   AxisStore[5].Axis[1..15].Pos26.Reached := FALSE;
   AxisStore[6].Axis[1..15].Pos26.Reached := FALSE;
   AxisStore[7].Axis[1..15].Pos26.Reached := FALSE;
   AxisStore[8].Axis[1..15].Pos26.Reached := FALSE;
   AxisStore[9].Axis[1..15].Pos26.Reached := FALSE;
   AxisStore[10].Axis[1..15].Pos26.Reached := FALSE;
   AxisStore[11].Axis[1..15].Pos26.Reached := FALSE;
   AxisStore[12].Axis[1..15].Pos26.Reached := FALSE;
   AxisStore[13].Axis[1..15].Pos26.Reached := FALSE;
   AxisStore[14].Axis[1..15].Pos26.Reached := FALSE;
   AxisStore[15].Axis[1..15].Pos26.Reached := FALSE;
   AxisStore[1].Axis[1..15].Pos27.Position := 0.0;
   AxisStore[2].Axis[1..15].Pos27.Position := 0.0;
   AxisStore[3].Axis[1..15].Pos27.Position := 0.0;
   AxisStore[4].Axis[1..15].Pos27.Position := 0.0;
   AxisStore[5].Axis[1..15].Pos27.Position := 0.0;
   AxisStore[6].Axis[1..15].Pos27.Position := 0.0;
   AxisStore[7].Axis[1..15].Pos27.Position := 0.0;
   AxisStore[8].Axis[1..15].Pos27.Position := 0.0;
   AxisStore[9].Axis[1..15].Pos27.Position := 0.0;
   AxisStore[10].Axis[1..15].Pos27.Position := 0.0;
   AxisStore[11].Axis[1..15].Pos27.Position := 0.0;
   AxisStore[12].Axis[1..15].Pos27.Position := 0.0;
   AxisStore[13].Axis[1..15].Pos27.Position := 0.0;
   AxisStore[14].Axis[1..15].Pos27.Position := 0.0;
   AxisStore[15].Axis[1..15].Pos27.Position := 0.0;
   AxisStore[1].Axis[1..15].Pos27.Speed := 0;
   AxisStore[2].Axis[1..15].Pos27.Speed := 0;
   AxisStore[3].Axis[1..15].Pos27.Speed := 0;
   AxisStore[4].Axis[1..15].Pos27.Speed := 0;
   AxisStore[5].Axis[1..15].Pos27.Speed := 0;
   AxisStore[6].Axis[1..15].Pos27.Speed := 0;
   AxisStore[7].Axis[1..15].Pos27.Speed := 0;
   AxisStore[8].Axis[1..15].Pos27.Speed := 0;
   AxisStore[9].Axis[1..15].Pos27.Speed := 0;
   AxisStore[10].Axis[1..15].Pos27.Speed := 0;
   AxisStore[11].Axis[1..15].Pos27.Speed := 0;
   AxisStore[12].Axis[1..15].Pos27.Speed := 0;
   AxisStore[13].Axis[1..15].Pos27.Speed := 0;
   AxisStore[14].Axis[1..15].Pos27.Speed := 0;
   AxisStore[15].Axis[1..15].Pos27.Speed := 0;
   AxisStore[1].Axis[1..15].Pos27.Reached := FALSE;
   AxisStore[2].Axis[1..15].Pos27.Reached := FALSE;
   AxisStore[3].Axis[1..15].Pos27.Reached := FALSE;
   AxisStore[4].Axis[1..15].Pos27.Reached := FALSE;
   AxisStore[5].Axis[1..15].Pos27.Reached := FALSE;
   AxisStore[6].Axis[1..15].Pos27.Reached := FALSE;
   AxisStore[7].Axis[1..15].Pos27.Reached := FALSE;
   AxisStore[8].Axis[1..15].Pos27.Reached := FALSE;
   AxisStore[9].Axis[1..15].Pos27.Reached := FALSE;
   AxisStore[10].Axis[1..15].Pos27.Reached := FALSE;
   AxisStore[11].Axis[1..15].Pos27.Reached := FALSE;
   AxisStore[12].Axis[1..15].Pos27.Reached := FALSE;
   AxisStore[13].Axis[1..15].Pos27.Reached := FALSE;
   AxisStore[14].Axis[1..15].Pos27.Reached := FALSE;
   AxisStore[15].Axis[1..15].Pos27.Reached := FALSE;
   AxisStore[1].Axis[1..15].Pos28.Position := 0.0;
   AxisStore[2].Axis[1..15].Pos28.Position := 0.0;
   AxisStore[3].Axis[1..15].Pos28.Position := 0.0;
   AxisStore[4].Axis[1..15].Pos28.Position := 0.0;
   AxisStore[5].Axis[1..15].Pos28.Position := 0.0;
   AxisStore[6].Axis[1..15].Pos28.Position := 0.0;
   AxisStore[7].Axis[1..15].Pos28.Position := 0.0;
   AxisStore[8].Axis[1..15].Pos28.Position := 0.0;
   AxisStore[9].Axis[1..15].Pos28.Position := 0.0;
   AxisStore[10].Axis[1..15].Pos28.Position := 0.0;
   AxisStore[11].Axis[1..15].Pos28.Position := 0.0;
   AxisStore[12].Axis[1..15].Pos28.Position := 0.0;
   AxisStore[13].Axis[1..15].Pos28.Position := 0.0;
   AxisStore[14].Axis[1..15].Pos28.Position := 0.0;
   AxisStore[15].Axis[1..15].Pos28.Position := 0.0;
   AxisStore[1].Axis[1..15].Pos28.Speed := 0;
   AxisStore[2].Axis[1..15].Pos28.Speed := 0;
   AxisStore[3].Axis[1..15].Pos28.Speed := 0;
   AxisStore[4].Axis[1..15].Pos28.Speed := 0;
   AxisStore[5].Axis[1..15].Pos28.Speed := 0;
   AxisStore[6].Axis[1..15].Pos28.Speed := 0;
   AxisStore[7].Axis[1..15].Pos28.Speed := 0;
   AxisStore[8].Axis[1..15].Pos28.Speed := 0;
   AxisStore[9].Axis[1..15].Pos28.Speed := 0;
   AxisStore[10].Axis[1..15].Pos28.Speed := 0;
   AxisStore[11].Axis[1..15].Pos28.Speed := 0;
   AxisStore[12].Axis[1..15].Pos28.Speed := 0;
   AxisStore[13].Axis[1..15].Pos28.Speed := 0;
   AxisStore[14].Axis[1..15].Pos28.Speed := 0;
   AxisStore[15].Axis[1..15].Pos28.Speed := 0;
   AxisStore[1].Axis[1..15].Pos28.Reached := FALSE;
   AxisStore[2].Axis[1..15].Pos28.Reached := FALSE;
   AxisStore[3].Axis[1..15].Pos28.Reached := FALSE;
   AxisStore[4].Axis[1..15].Pos28.Reached := FALSE;
   AxisStore[5].Axis[1..15].Pos28.Reached := FALSE;
   AxisStore[6].Axis[1..15].Pos28.Reached := FALSE;
   AxisStore[7].Axis[1..15].Pos28.Reached := FALSE;
   AxisStore[8].Axis[1..15].Pos28.Reached := FALSE;
   AxisStore[9].Axis[1..15].Pos28.Reached := FALSE;
   AxisStore[10].Axis[1..15].Pos28.Reached := FALSE;
   AxisStore[11].Axis[1..15].Pos28.Reached := FALSE;
   AxisStore[12].Axis[1..15].Pos28.Reached := FALSE;
   AxisStore[13].Axis[1..15].Pos28.Reached := FALSE;
   AxisStore[14].Axis[1..15].Pos28.Reached := FALSE;
   AxisStore[15].Axis[1..15].Pos28.Reached := FALSE;
   AxisStore[1].Axis[1..15].Pos29.Position := 0.0;
   AxisStore[2].Axis[1..15].Pos29.Position := 0.0;
   AxisStore[3].Axis[1..15].Pos29.Position := 0.0;
   AxisStore[4].Axis[1..15].Pos29.Position := 0.0;
   AxisStore[5].Axis[1..15].Pos29.Position := 0.0;
   AxisStore[6].Axis[1..15].Pos29.Position := 0.0;
   AxisStore[7].Axis[1..15].Pos29.Position := 0.0;
   AxisStore[8].Axis[1..15].Pos29.Position := 0.0;
   AxisStore[9].Axis[1..15].Pos29.Position := 0.0;
   AxisStore[10].Axis[1..15].Pos29.Position := 0.0;
   AxisStore[11].Axis[1..15].Pos29.Position := 0.0;
   AxisStore[12].Axis[1..15].Pos29.Position := 0.0;
   AxisStore[13].Axis[1..15].Pos29.Position := 0.0;
   AxisStore[14].Axis[1..15].Pos29.Position := 0.0;
   AxisStore[15].Axis[1..15].Pos29.Position := 0.0;
   AxisStore[1].Axis[1..15].Pos29.Speed := 0;
   AxisStore[2].Axis[1..15].Pos29.Speed := 0;
   AxisStore[3].Axis[1..15].Pos29.Speed := 0;
   AxisStore[4].Axis[1..15].Pos29.Speed := 0;
   AxisStore[5].Axis[1..15].Pos29.Speed := 0;
   AxisStore[6].Axis[1..15].Pos29.Speed := 0;
   AxisStore[7].Axis[1..15].Pos29.Speed := 0;
   AxisStore[8].Axis[1..15].Pos29.Speed := 0;
   AxisStore[9].Axis[1..15].Pos29.Speed := 0;
   AxisStore[10].Axis[1..15].Pos29.Speed := 0;
   AxisStore[11].Axis[1..15].Pos29.Speed := 0;
   AxisStore[12].Axis[1..15].Pos29.Speed := 0;
   AxisStore[13].Axis[1..15].Pos29.Speed := 0;
   AxisStore[14].Axis[1..15].Pos29.Speed := 0;
   AxisStore[15].Axis[1..15].Pos29.Speed := 0;
   AxisStore[1].Axis[1..15].Pos29.Reached := FALSE;
   AxisStore[2].Axis[1..15].Pos29.Reached := FALSE;
   AxisStore[3].Axis[1..15].Pos29.Reached := FALSE;
   AxisStore[4].Axis[1..15].Pos29.Reached := FALSE;
   AxisStore[5].Axis[1..15].Pos29.Reached := FALSE;
   AxisStore[6].Axis[1..15].Pos29.Reached := FALSE;
   AxisStore[7].Axis[1..15].Pos29.Reached := FALSE;
   AxisStore[8].Axis[1..15].Pos29.Reached := FALSE;
   AxisStore[9].Axis[1..15].Pos29.Reached := FALSE;
   AxisStore[10].Axis[1..15].Pos29.Reached := FALSE;
   AxisStore[11].Axis[1..15].Pos29.Reached := FALSE;
   AxisStore[12].Axis[1..15].Pos29.Reached := FALSE;
   AxisStore[13].Axis[1..15].Pos29.Reached := FALSE;
   AxisStore[14].Axis[1..15].Pos29.Reached := FALSE;
   AxisStore[15].Axis[1..15].Pos29.Reached := FALSE;
   AxisStore[1].Axis[1..15].Pos30.Position := 0.0;
   AxisStore[2].Axis[1..15].Pos30.Position := 0.0;
   AxisStore[3].Axis[1..15].Pos30.Position := 0.0;
   AxisStore[4].Axis[1..15].Pos30.Position := 0.0;
   AxisStore[5].Axis[1..15].Pos30.Position := 0.0;
   AxisStore[6].Axis[1..15].Pos30.Position := 0.0;
   AxisStore[7].Axis[1..15].Pos30.Position := 0.0;
   AxisStore[8].Axis[1..15].Pos30.Position := 0.0;
   AxisStore[9].Axis[1..15].Pos30.Position := 0.0;
   AxisStore[10].Axis[1..15].Pos30.Position := 0.0;
   AxisStore[11].Axis[1..15].Pos30.Position := 0.0;
   AxisStore[12].Axis[1..15].Pos30.Position := 0.0;
   AxisStore[13].Axis[1..15].Pos30.Position := 0.0;
   AxisStore[14].Axis[1..15].Pos30.Position := 0.0;
   AxisStore[15].Axis[1..15].Pos30.Position := 0.0;
   AxisStore[1].Axis[1..15].Pos30.Speed := 0;
   AxisStore[2].Axis[1..15].Pos30.Speed := 0;
   AxisStore[3].Axis[1..15].Pos30.Speed := 0;
   AxisStore[4].Axis[1..15].Pos30.Speed := 0;
   AxisStore[5].Axis[1..15].Pos30.Speed := 0;
   AxisStore[6].Axis[1..15].Pos30.Speed := 0;
   AxisStore[7].Axis[1..15].Pos30.Speed := 0;
   AxisStore[8].Axis[1..15].Pos30.Speed := 0;
   AxisStore[9].Axis[1..15].Pos30.Speed := 0;
   AxisStore[10].Axis[1..15].Pos30.Speed := 0;
   AxisStore[11].Axis[1..15].Pos30.Speed := 0;
   AxisStore[12].Axis[1..15].Pos30.Speed := 0;
   AxisStore[13].Axis[1..15].Pos30.Speed := 0;
   AxisStore[14].Axis[1..15].Pos30.Speed := 0;
   AxisStore[15].Axis[1..15].Pos30.Speed := 0;
   AxisStore[1].Axis[1..15].Pos30.Reached := FALSE;
   AxisStore[2].Axis[1..15].Pos30.Reached := FALSE;
   AxisStore[3].Axis[1..15].Pos30.Reached := FALSE;
   AxisStore[4].Axis[1..15].Pos30.Reached := FALSE;
   AxisStore[5].Axis[1..15].Pos30.Reached := FALSE;
   AxisStore[6].Axis[1..15].Pos30.Reached := FALSE;
   AxisStore[7].Axis[1..15].Pos30.Reached := FALSE;
   AxisStore[8].Axis[1..15].Pos30.Reached := FALSE;
   AxisStore[9].Axis[1..15].Pos30.Reached := FALSE;
   AxisStore[10].Axis[1..15].Pos30.Reached := FALSE;
   AxisStore[11].Axis[1..15].Pos30.Reached := FALSE;
   AxisStore[12].Axis[1..15].Pos30.Reached := FALSE;
   AxisStore[13].Axis[1..15].Pos30.Reached := FALSE;
   AxisStore[14].Axis[1..15].Pos30.Reached := FALSE;
   AxisStore[15].Axis[1..15].Pos30.Reached := FALSE;
END_DATA_BLOCK

DATA_BLOCK "ST10_RecipeActiveDB"   // DB1064
{ S7_Optimized_Access := 'FALSE' }
// stored: AutoNumber false
   VAR RETAIN
      Recipe : Struct   // System Defined=
         RecipeTag : String[50];   // 配方名称ID
         RecordName : String[50];   // 数据记录名称
         PreConfigType : String[50];   // 待切换数据记录名称
         Pulse : Bool;
         Trigger : Bool;   // 配方切换触发
         PosEdg : Bool;
         Alarm : Bool;
         Ret : Bool;
         Equal : Bool;
         Pls : Bool;
         "time" : Int;
         Spare : Array[0..38] of Byte;
         DataRecord_TransferStatus : Int;   // 数据记录传送状态
      END_STRUCT;
      ParameterElement : Struct
         TypeName : String[50];   // System Defined=
         TypeID : Int;   // System define= product type for parameters of servo ,press and so on
         FixtureID : Array[0..5] of Int;
         FestoAxis : "RecipeAxis";
         PressRgramNo { S7_SetPoint := 'True'} : Array[0..60] of DInt;
         ProcessParameter { S7_SetPoint := 'True'} : "MEStoPLC_RecipeData_OP220";
      END_STRUCT;
   END_VAR
BEGIN
END_DATA_BLOCK

DATA_BLOCK "ST10_RecipeDB"   // DB1062
{ S7_Optimized_Access := 'FALSE' }
// stored: AutoNumber false
   VAR RETAIN
      Recipe : Struct   // System Defined=
         RecipeTag : String[50] := 'RecipeST10';   // 配方名称ID / System Defined=
         RecordName : String[50] := 'Product_1';   // 数据记录名称 / 配方名称ID
         PreConfigType : String[50] := 'Product_1';   // 待切换数据记录名称 / 数据记录名称
         Pulse : Bool := FALSE;   // 待切换数据记录名称
         Trigger : Bool := FALSE;   // 配方切换触发
         PosEdg : Bool := FALSE;   // 配方切换触发
         Alarm : Bool := FALSE;
         Ret : Bool := FALSE;
         Equal : Bool := TRUE;   // 换型OK标志位
         Pls : Bool := FALSE;   // 换型OK标志位
         "time" : Int := 0;
         Spare : Array[0..38] of Byte;
         DataRecord_TransferStatus : Int := 0;   // 数据记录传送状态
      END_STRUCT;
      ParameterElement : Struct
         TypeName : String[50] := 'Product_1';   // System Defined=
         TypeID : USInt := 1;   // System define= product type for parameters of servo ,press and so on
         FixtureID : Array[1..16] of Byte;
         A1_TableFixtureCode : Array[0..10] of String[128];   // 激光刻印程序号
         A2_TableFixtureCode : Array[0..10] of String[128];   // 贴标10号垂直气缸是否去工作位
         A1RingUnloadingFixtureCode : String[128] := 'SZ23055-OP010-E-Compresspr-ring1 cutting tool';
         E1LoadingNGFixtureCode : String[128] := 'SZ23055-OP010-E-Compressor-Left NG tooling-1';
         ShaftScanFixtureCode : String[128] := 'SZ23055-OP010-E-Compressor-shaft Rotating scanning tooling-1';
         B1PressFixtureCode : String[128] := 'SZ23055-OP010-E-Compressor-ring1 Below Positioning fixture -1';
         CGlueFixtureCode : String[128] := 'SZ23055-OP010-E-Compressor-Point adhesive tooling-1';
         B1PressCylFixtureCode : String[128] := 'SZ23055-OP010-E-Compressor-ring1 Upper pressing fixture-1';
         A2RingUnloadingFixtureCode : String[128] := 'SZ23055-OP010-E-Compresspr-ring2 cutting tool';
         E2UnloadingNGFixtureCode : String[128] := 'SZ23055-OP010-E-Compressor-Right NG tooling-1';
         B2PressFixtureCode : String[128] := 'SZ23055-OP010-E-Compressor-ring2 Below Positioning fixture -1';
         CGlueNGFixtureCode : String[128] := 'SZ23055-OP010-E-Compressor-NG middle shift tooling-1';
         B2PressCylFixtureCode : String[128] := 'SZ23055-OP010-E-Compressor-ring2 Upper pressing fixture-1';
         R1GripperFixtureCode : Array[0..6] of String[128];
         R2GripperFixtureCode : Array[0..6] of String[128];
         R3GripperFixtureCode : Array[0..6] of String[128];
         B1PressProgram : Int := 1;
         B2PressProgram : Int := 1;
         CGlueShaftIV3Program_1 : Word := 16#0001;
         CGlueShaftIV3Program_2 : Word := 16#0002;
         CGlueShaftIV3Program_3 : Word := 16#0003;
         CGlueShaftIV3Program_4 : Word := 16#0004;
         CGlueMagnetIV3Program : Word := 16#0001;
         CGlueProgram : Int := 1;
      END_STRUCT;
   END_VAR
BEGIN
   Recipe.Spare[0..38] := 16#00;
   ParameterElement.FixtureID[1] := 16#00;   // 工装编号
   ParameterElement.FixtureID[2..16] := 16#00;
   ParameterElement.A1_TableFixtureCode[0] := '';
   ParameterElement.A1_TableFixtureCode[1] := 'SZ23055-OP010-E-Compressor-ring1 Loading tooling-1';
   ParameterElement.A1_TableFixtureCode[2] := 'SZ23055-OP010-E-Compressor-ring1 Loading tooling-2';
   ParameterElement.A1_TableFixtureCode[3] := 'SZ23055-OP010-E-Compressor-ring1 Loading tooling-3';
   ParameterElement.A1_TableFixtureCode[4] := 'SZ23055-OP010-E-Compressor-ring1 Loading tooling-4';
   ParameterElement.A1_TableFixtureCode[5] := 'SZ23055-OP010-E-Compressor-ring1 Loading tooling-5';
   ParameterElement.A1_TableFixtureCode[6] := 'SZ23055-OP010-E-Compressor-ring1 Loading tooling-6';
   ParameterElement.A1_TableFixtureCode[7] := 'SZ23055-OP010-E-Compressor-ring1 Loading tooling-7';
   ParameterElement.A1_TableFixtureCode[8] := 'SZ23055-OP010-E-Compressor-ring1 Loading tooling-8';
   ParameterElement.A1_TableFixtureCode[9..10] := '';
   ParameterElement.A2_TableFixtureCode[0] := '';
   ParameterElement.A2_TableFixtureCode[1] := 'SZ23055-OP010-E-Compressor-ring2 Loading tooling-1';
   ParameterElement.A2_TableFixtureCode[2] := 'SZ23055-OP010-E-Compressor-ring2 Loading tooling-2';
   ParameterElement.A2_TableFixtureCode[3] := 'SZ23055-OP010-E-Compressor-ring2 Loading tooling-3';
   ParameterElement.A2_TableFixtureCode[4] := 'SZ23055-OP010-E-Compressor-ring2 Loading tooling-4';
   ParameterElement.A2_TableFixtureCode[5] := 'SZ23055-OP010-E-Compressor-ring2 Loading tooling-5';
   ParameterElement.A2_TableFixtureCode[6] := 'SZ23055-OP010-E-Compressor-ring2 Loading tooling-6';
   ParameterElement.A2_TableFixtureCode[7] := 'SZ23055-OP010-E-Compressor-ring2 Loading tooling-7';
   ParameterElement.A2_TableFixtureCode[8] := 'SZ23055-OP010-E-Compressor-ring2 Loading tooling-8';
   ParameterElement.A2_TableFixtureCode[9..10] := '';
   ParameterElement.R1GripperFixtureCode[0] := '';
   ParameterElement.R1GripperFixtureCode[1] := 'SZ23055-OP010-E-Compressor-robot1 ring1 Left clamping jaw tooling-1';
   ParameterElement.R1GripperFixtureCode[2] := 'SZ23055-OP010-E-Compressor-robot1 ring1 Right clamping jaw tooling-2';
   ParameterElement.R1GripperFixtureCode[3] := 'SZ23055-OP010-E-Compressor-robot1 shaft Left clamping jaw tooling-1';
   ParameterElement.R1GripperFixtureCode[4] := 'SZ23055-OP010-E-Compressor-robot1 shaft Right clamping jaw tooling-2';
   ParameterElement.R1GripperFixtureCode[5..6] := '';
   ParameterElement.R2GripperFixtureCode[0] := '';
   ParameterElement.R2GripperFixtureCode[1] := 'SZ23055-OP010-E-Compressor-robot2 shaft Right clamping jaw tooling-2';
   ParameterElement.R2GripperFixtureCode[2] := 'SZ23055-OP010-E-Compressor-robot2 shaft Left clamping jaw tooling-1';
   ParameterElement.R2GripperFixtureCode[3] := 'SZ23055-OP010-E-Compressor-robot2 magnet Left clamping jaw tooling-1';
   ParameterElement.R2GripperFixtureCode[4] := 'SZ23055-OP010-E-Compressor-robot2 magnet Right clamping jaw tooling-2';
   ParameterElement.R2GripperFixtureCode[5..6] := '';
   ParameterElement.R3GripperFixtureCode[0] := '';
   ParameterElement.R3GripperFixtureCode[1] := 'SZ23055-OP010-E-Compressor-robot3 ring2 Right clamping jaw tooling-2';
   ParameterElement.R3GripperFixtureCode[2] := 'SZ23055-OP010-E-Compressor-robot3 ring2 Left clamping jaw tooling-1';
   ParameterElement.R3GripperFixtureCode[3] := 'SZ23055-OP010-E-Compressor-robot3 shaft Left clamping jaw tooling-1';
   ParameterElement.R3GripperFixtureCode[4] := 'SZ23055-OP010-E-Compressor-robot3 shaft Right clamping jaw tooling-2';
   ParameterElement.R3GripperFixtureCode[5..6] := '';
END_DATA_BLOCK

DATA_BLOCK "ST10_RecipeDB_HMI"   // DB1079
{ S7_Optimized_Access := 'FALSE' }
// stored: AutoNumber false
   VAR RETAIN
      Recipe : Struct   // System Defined=
         RecipeTag : String[50] := 'RecipeST10';   // 配方名称ID / System Defined=
         RecordName : String[50] := 'Product_1';   // 数据记录名称 / 配方名称ID
         PreConfigType : String[50] := 'Product_1';   // 待切换数据记录名称 / 数据记录名称
         Pulse : Bool := FALSE;   // 待切换数据记录名称
         Trigger : Bool := FALSE;   // 配方切换触发
         PosEdg : Bool := TRUE;   // 配方切换触发
         Alarm : Bool := FALSE;
         Ret : Bool := FALSE;
         Equal : Bool := TRUE;   // 换型OK标志位
         Pls : Bool := FALSE;   // 换型OK标志位
         "time" : Int := 0;
         Spare : Array[0..38] of Byte;
         DataRecord_TransferStatus : Int := 0;   // 数据记录传送状态
      END_STRUCT;
      ParameterElement : Struct
         TypeName : String[50] := 'Product_1';   // System Defined=
         TypeID : USInt := 1;   // System define= product type for parameters of servo ,press and so on
         FixtureID : Array[1..16] of Byte;
         A1_TableFixtureCode : Array[0..10] of String[128];   // 激光刻印程序号
         A2_TableFixtureCode : Array[0..10] of String[128];   // 贴标10号垂直气缸是否去工作位
         A1RingUnloadingFixtureCode : String[128] := 'F2';
         E1LoadingNGFixtureCode : String[128] := 'SZ23055-OP010-E-Compressor-Left NG tooling-1';
         ShaftScanFixtureCode : String[128] := 'SZ23055-OP010-E-Compressor-shaft Rotating scanning tooling-1';
         B1PressFixtureCode : String[128] := 'SZ23055-OP010-E-Compressor-ring1 Below Positioning fixture -1';
         CGlueFixtureCode : String[128] := 'SZ23055-OP010-E-Compressor-Point adhesive tooling-1';
         B1PressCylFixtureCode : String[128] := 'SZ23055-OP010-E-Compressor-ring1 Upper pressing fixture-1';
         A2RingUnloadingFixtureCode : String[128] := 'F12';
         E2UnloadingNGFixtureCode : String[128] := 'SZ23055-OP010-E-Compressor-Right NG tooling-1';
         B2PressFixtureCode : String[128] := 'SZ23055-OP010-E-Compressor-ring2 Below Positioning fixture -1';
         CGlueNGFixtureCode : String[128] := 'SZ23055-OP010-E-Compressor-NG middle shift tooling-1';
         B2PressCylFixtureCode : String[128] := 'SZ23055-OP010-E-Compressor-ring1 Upper pressing fixture-1';
         R1GripperFixtureCode : Array[0..6] of String[128];
         R2GripperFixtureCode : Array[0..6] of String[128];
         R3GripperFixtureCode : Array[0..6] of String[128];
         B1PressProgram : Int := 1;
         B2PressProgram : Int := 1;
         CGlueShaftIV3Program_1 : Word := 16#0001;
         CGlueShaftIV3Program_2 : Word := 16#0002;
         CGlueShaftIV3Program_3 : Word := 16#0003;
         CGlueShaftIV3Program_4 : Word := 16#0004;
         CGlueMagnetIV3Program : Word := 16#0001;
         CGlueProgram : Int := 1;
      END_STRUCT;
   END_VAR
BEGIN
   Recipe.Spare[0..38] := 16#00;
   ParameterElement.FixtureID[1] := 16#00;   // 工装编号
   ParameterElement.FixtureID[2..16] := 16#00;
   ParameterElement.A1_TableFixtureCode[0] := '';
   ParameterElement.A1_TableFixtureCode[1] := 'SZ23055-OP010-E-Compressor-ring1 Loading tooling-1';
   ParameterElement.A1_TableFixtureCode[2] := 'SZ23055-OP010-E-Compressor-ring1 Loading tooling-2';
   ParameterElement.A1_TableFixtureCode[3] := 'SZ23055-OP010-E-Compressor-ring1 Loading tooling-3';
   ParameterElement.A1_TableFixtureCode[4] := 'SZ23055-OP010-E-Compressor-ring1 Loading tooling-4';
   ParameterElement.A1_TableFixtureCode[5] := 'SZ23055-OP010-E-Compressor-ring1 Loading tooling-5';
   ParameterElement.A1_TableFixtureCode[6] := 'SZ23055-OP010-E-Compressor-ring1 Loading tooling-6';
   ParameterElement.A1_TableFixtureCode[7] := 'SZ23055-OP010-E-Compressor-ring1 Loading tooling-7';
   ParameterElement.A1_TableFixtureCode[8] := 'SZ23055-OP010-E-Compressor-ring1 Loading tooling-8';
   ParameterElement.A1_TableFixtureCode[9..10] := '';
   ParameterElement.A2_TableFixtureCode[0] := '';
   ParameterElement.A2_TableFixtureCode[1] := 'SZ23055-OP010-E-Compressor-ring2 Loading tooling-1';
   ParameterElement.A2_TableFixtureCode[2] := 'SZ23055-OP010-E-Compressor-ring2 Loading tooling-2';
   ParameterElement.A2_TableFixtureCode[3] := 'SZ23055-OP010-E-Compressor-ring2 Loading tooling-3';
   ParameterElement.A2_TableFixtureCode[4] := 'SZ23055-OP010-E-Compressor-ring2 Loading tooling-4';
   ParameterElement.A2_TableFixtureCode[5] := 'SZ23055-OP010-E-Compressor-ring2 Loading tooling-5';
   ParameterElement.A2_TableFixtureCode[6] := 'SZ23055-OP010-E-Compressor-ring2 Loading tooling-6';
   ParameterElement.A2_TableFixtureCode[7] := 'SZ23055-OP010-E-Compressor-ring2 Loading tooling-7';
   ParameterElement.A2_TableFixtureCode[8] := 'SZ23055-OP010-E-Compressor-ring2 Loading tooling-8';
   ParameterElement.A2_TableFixtureCode[9..10] := '';
   ParameterElement.R1GripperFixtureCode[0] := '';
   ParameterElement.R1GripperFixtureCode[1] := 'SZ23055-OP010-E-Compressor-robot1 ring1 Left clamping jaw tooling-1';
   ParameterElement.R1GripperFixtureCode[2] := 'SZ23055-OP010-E-Compressor-robot1 ring1 Right clamping jaw tooling-2';
   ParameterElement.R1GripperFixtureCode[3] := 'SZ23055-OP010-E-Compressor-robot1 shaft Left clamping jaw tooling-1';
   ParameterElement.R1GripperFixtureCode[4] := 'SZ23055-OP010-E-Compressor-robot1 shaft Right clamping jaw tooling-2';
   ParameterElement.R1GripperFixtureCode[5..6] := '';
   ParameterElement.R2GripperFixtureCode[0] := '';
   ParameterElement.R2GripperFixtureCode[1] := 'SZ23055-OP010-E-Compressor-robot2 shaft Right clamping jaw tooling-2';
   ParameterElement.R2GripperFixtureCode[2] := 'SZ23055-OP010-E-Compressor-robot2 shaft Left clamping jaw tooling-1';
   ParameterElement.R2GripperFixtureCode[3] := 'SZ23055-OP010-E-Compressor-robot2 magnet Left clamping jaw tooling-1';
   ParameterElement.R2GripperFixtureCode[4] := 'SZ23055-OP010-E-Compressor-robot2 magnet Right clamping jaw tooling-2';
   ParameterElement.R2GripperFixtureCode[5..6] := '';
   ParameterElement.R3GripperFixtureCode[0] := '';
   ParameterElement.R3GripperFixtureCode[1] := 'SZ23055-OP010-E-Compressor-robot3 ring2 Right clamping jaw tooling-2';
   ParameterElement.R3GripperFixtureCode[2] := 'SZ23055-OP010-E-Compressor-robot3 ring2 Left clamping jaw tooling-1';
   ParameterElement.R3GripperFixtureCode[3] := 'SZ23055-OP010-E-Compressor-robot3 shaft Left clamping jaw tooling-1';
   ParameterElement.R3GripperFixtureCode[4] := 'SZ23055-OP010-E-Compressor-robot3 shaft Right clamping jaw tooling-2';
   ParameterElement.R3GripperFixtureCode[5..6] := '';
END_DATA_BLOCK

DATA_BLOCK "ST10_PMCountCycleTime"   // DB1061
{ S7_Optimized_Access := 'FALSE' }
// stored: AutoNumber false
   VAR
      PM : Array[1..30] of "RCS_CountCycleTime_V1";
      PM_Num : Int;
   END_VAR
BEGIN
END_DATA_BLOCK

DATA_BLOCK "MES_CheckControl"   // DB2361
{ S7_Optimized_Access := 'FALSE' }
// stored: AutoNumber false
   VAR
      ST1MesCheckIn : Bool;
      ST1MesCheckOut : Bool;
      ST2MesCheckIn : Bool;
      ST2MesCheckOut : Bool;
      ST3MesCheckIn : Bool;
      ST3MesCheckOut : Bool;
      ST4MesCheckIn : Bool;
      ST4MesCheckOut : Bool;
      Station1 : Struct
         CheckInRequest : Bool;
         CheckResultRequest : Bool;
      END_STRUCT;
      Station2 : Struct
         CheckInRequest : Bool;
         CheckResultRequest : Bool;
      END_STRUCT;
      Station3 : Struct
         CheckInRequest : Bool;
         CheckResultRequest : Bool;
      END_STRUCT;
      Station4 : Struct
         CheckInRequest : Bool;
         CheckResultRequest : Bool;
      END_STRUCT;
      Station5 : Struct
         CheckInRequest : Bool;
         CheckResultRequest : Bool;
      END_STRUCT;
      Station6 : Struct
         CheckInRequest : Bool;
         CheckResultRequest : Bool;
      END_STRUCT;
      Station7 : Struct
         CheckInRequest : Bool;
         CheckResultRequest : Bool;
      END_STRUCT;
   END_VAR
BEGIN
END_DATA_BLOCK

DATA_BLOCK "MEStoPLC"   // DB501
{ S7_Optimized_Access := 'FALSE' }
// stored: AutoNumber false
   VAR
      "MES.Load_Station1PartOK" : Bool;   // 激光打标过站查询事件反馈 OK
      "MES.Load_Station1PartNG" : Bool;   // 激光打标过站查询事件反馈 NG
      "MES.Load_Station1ReqMesDone" : Bool;   // 激光打标过站查询事件反馈 DONE
      Spare_1 : Bool;
      "MES.Load_Station2PartOK" : Bool;
      "MES.Load_Station2PartNG" : Bool;
      "MES.Load_Station2ReqMesDone" : Bool;
      Spare_2 : Bool;
      "MES.Load_Station3PartOK" : Bool;   // 读码贴标过站查询事件反馈 OK
      "MES.Load_Station3PartNG" : Bool;   // 读码贴标过站查询事件反馈 NG
      "MES.Load_Station3ReqMesDone" : Bool;   // 读码贴标过站查询事件反馈 DONE
      Spare_3 : Bool;
      "MES.Load_Station4PartOK" : Bool;
      "MES.Load_Station4PartNG" : Bool;
      "MES.Load_Station4ReqMesDone" : Bool;
      Spare_4 : Bool;
      "MES.Load_Station5PartOK" : Bool;
      "MES.Load_Station5PartNG" : Bool;
      "MES.Load_Station5ReqMesDone" : Bool;
      Spare_5 : Bool;
      "MES.Load_Station6PartOK" : Bool;
      "MES.Load_Station6PartNG" : Bool;
      "MES.Load_Station6ReqMesDone" : Bool;
      Spare_6 : Bool;
      "MES.Load_Station7PartOK" : Bool;
      "MES.Load_Station7PartNG" : Bool;
      "MES.Load_Station7ReqMesDone" : Bool;
      Spare_7 : Bool;
      "MES.Load_Station8PartOK" : Bool;
      "MES.Load_Station8PartNG" : Bool;
      "MES.Load_Station8ReqMesDone" : Bool;
      Spare_8 : Bool;
      Spare_9 : Bool;
      Static_3 : Bool;
      "MES.Load_SubPart1OK" : Bool;
      "MES.Load_SubPart1tNG" : Bool;
      "MES.Load_SubPart1ReqMesDone" : Bool;
      Spare_10 : Bool;
      "MES.Load_SubPart2OK" : Bool;
      "MES.Load_SubPart2tNG" : Bool;
      "MES.Load_SubPart2ReqMesDone" : Bool;
      Spare_11 : Bool;
      "MES.Load_SubPart3OK" : Bool;
      "MES.Load_SubPart3tNG" : Bool;
      "MES.Load_SubPart3ReqMesDone" : Bool;
      Spare_12 : Bool;
      "MES.Load_SubPart4OK" : Bool;
      "MES.Load_SubPart4tNG" : Bool;
      "MES.Load_SubPart4ReqMesDone" : Bool;
      Spare_13 : Bool;
      "MES.Load_SubPart5OK" : Bool;
      "MES.Load_SubPart5tNG" : Bool;
      "MES.Load_SubPart5ReqMesDone" : Bool;
      Spare_14 : Bool;
      "MES.Load_SubPart6OK" : Bool;
      "MES.Load_SubPart6tNG" : Bool;
      "MES.Load_SubPart6ReqMesDone" : Bool;
      Spare_15 : Bool;
      "MES.Load_SubPart7OK" : Bool;
      "MES.Load_SubPart7tNG" : Bool;
      "MES.Load_SubPart7ReqMesDone" : Bool;
      Spare_16 : Bool;
      "MES.Load_SubPart8OK" : Bool;
      "MES.Load_SubPart8tNG" : Bool;
      "MES.Load_SubPart8ReqMesDone" : Bool;
      Spare : Bool;
      Spare_17 : Bool;
      "MES.Load_ResultsStored1OK" : Bool;
      "MES.Load_ResultsStored1NG" : Bool;
      "MES.Load_ResultsStored1ReqMesDone" : Bool;
      Spare_18 : Bool;
      "MES.Load_ResultsStored2OK" : Bool;
      "MES.Load_ResultsStored2NG" : Bool;
      "MES.Load_ResultsStored2ReqMesDone" : Bool;
      Spare_19 : Bool;
      "MES.Load_ResultsStored3OK" : Bool;
      "MES.Load_ResultsStored3NG" : Bool;
      "MES.Load_ResultsStored3ReqMesDone" : Bool;
      Spare_20 : Bool;
      "MES.Load_ResultsStored4OK" : Bool;
      "MES.Load_ResultsStored4NG" : Bool;
      "MES.Load_ResultsStored4ReqMesDone" : Bool;
      Spare_21 : Bool;
      "MES.Load_ResultsStored5OK" : Bool;
      "MES.Load_ResultsStored5NG" : Bool;
      "MES.Load_ResultsStored5ReqMesDone" : Bool;
      Spare_22 : Bool;
      "MES.Load_ResultsStored6OK" : Bool;
      "MES.Load_ResultsStored6NG" : Bool;
      "MES.Load_ResultsStored6ReqMesDone" : Bool;
      Spare_23 : Bool;
      "MES.Load_ResultsStored7OK" : Bool;
      "MES.Load_ResultsStored7NG" : Bool;
      "MES.Load_ResultsStored7ReqMesDone" : Bool;
      Spare_24 : Bool;
      "MES.Load_ResultsStored8OK" : Bool;
      "MES.Load_ResultsStored8NG" : Bool;
      "MES.Load_ResultsStored8ReqMesDone" : Bool;
      "MES.Load_StoveCheckInOk" : Bool;
      Static_1 : Bool;
      Spare_26 : Bool;
      Spare_27 : Bool;
      Spare_28 : Bool;
      Spare_29 : Bool;
      Spare_30 : Bool;
      Spare_31 : Bool;
      Spare_32 : Bool;
      Spare_33 : Bool;
      "MES.Unload_ResultsStored1OK" : Bool;
      "MES.Unload_ResultsStored1NG" : Bool;
      "MES.Unload_ResultsStored1ReqMesDone" : Bool;
      Spare_34 : Bool;
      "MES.Unload_ResultsStored2OK" : Bool;
      "MES.Unload_ResultsStored2NG" : Bool;
      "MES.Unload_ResultsStored2ReqMesDone" : Bool;
      Spare_35 : Bool;
      "MES.Unload_ResultsStored3OK" : Bool;
      "MES.Unload_ResultsStored3NG" : Bool;
      "MES.Unload_ResultsStored3ReqMesDone" : Bool;
      Spare_36 : Bool;
      "MES.Unload_ResultsStored4OK" : Bool;
      "MES.Unload_ResultsStored4NG" : Bool;
      "MES.Unload_ResultsStored4ReqMesDone" : Bool;
      Spare_37 : Bool;
      "MES.Unload_ResultsStored5OK" : Bool;
      "MES.Unload_ResultsStored5NG" : Bool;
      "MES.Unload_ResultsStored5ReqMesDone" : Bool;
      Spare_38 : Bool;
      "MES.Unload_ResultsStored6OK" : Bool;
      "MES.Unload_ResultsStored6NG" : Bool;
      "MES.Unload_ResultsStored6ReqMesDone" : Bool;
      Spare_39 : Bool;
      "MES.Unload_ResultsStored7OK" : Bool;
      "MES.Unload_ResultsStored7NG" : Bool;
      "MES.Unload_ResultsStored7ReqMesDone" : Bool;
      Spare_40 : Bool;
      "MES.Unload_ResultsStored8OK" : Bool;
      "MES.Unload_ResultsStored8NG" : Bool;
      "MES.Unload_ResultsStored8ReqMesDone" : Bool;
      Spare_41 : Bool;
      "MES.HeartbeatSignal" : Bool;
   END_VAR
BEGIN
END_DATA_BLOCK

DATA_BLOCK "PLCtoMES"   // DB500
{ S7_Optimized_Access := 'FALSE' }
// stored: AutoNumber false
   VAR
      "PLC.Load_Station1ChickInReq" : Bool;   // 本站工位1打标工位主零件RFID码读出，请求查询
      "PLC.Load_Station2ChickInReq" : Bool;   // 本站工位2贴标工位主零件RFID码读出，请求查询
      "PLC.Load_Station3ChickInReq" : Bool;   // Spare
      "PLC.Load_Station4ChickInReq" : Bool;   // Spare
      "PLC.Load_Station5ChickInReq" : Bool;   // Spare
      "PLC.Load_Station6ChickInReq" : Bool;   // Spare
      "PLC.Load_Station7ChickInReq" : Bool;   // Spare
      "PLC.Load_Station8ChickInReq" : Bool;   // Spare
      "PLC.Load_StoveCheckIn" : Bool;   // 子零件1码读出，请求查询
      Spare_11 : Bool;   // Spare
      Spare_12 : Bool;   // Spare
      Spare_13 : Bool;   // Spare
      Spare_14 : Bool;   // Spare
      Spare_15 : Bool;   // Spare
      Spare_16 : Bool;   // Spare
      Spare_17 : Bool;   // Spare
      Spare_18 : Bool;   // 手持扫码枪1上料查询触发
      Spare_19 : Bool;   // Spare
      Spare_20 : Bool;   // Spare
      Spare_21 : Bool;   // Spare
      Spare_22 : Bool;   // Spare
      Spare_23 : Bool;   // Spare
      Spare_24 : Bool;   // Spare
      Spare_25 : Bool;   // Spare
      Spare_1 : Byte;   // Spare
      Spare_2 : Bool;   // 请求下发打标数据触发
      Spare_3 : Bool;   // 二维码内容与主零件码比对请求
      Spare_4 : Bool;   // Spare
      Spare_5 : Bool;   // Spare
      Spare_6 : Bool;   // Spare
      Spare_7 : Bool;   // Spare
      Spare_8 : Bool;   // Spare
      Spare_9 : Bool;   // Spare
      Spare_10 : Bool;
      Static_2 : Bool;   // 本站工位1打标过程数据保存触发位
      "PLC.Unload_Station1DataSaveReq" : Bool;   // 本站工位2贴标过程数据保存触发位
      "PLC.Unload_Station2DataSaveReq" : Bool;   // Spare
      "PLC.Unload_Station3DataSaveReq" : Bool;   // Spare
      "PLC.Unload_Station4DataSaveReq" : Bool;   // Spare
      "PLC.Unload_Station5DataSaveReq" : Bool;   // Spare
      "PLC.Unload_Station6DataSaveReq" : Bool;   // Spare
      "PLC.Unload_Station7DataSaveReq" : Bool;   // Spare
      "PLC.Unload_Station8DataSaveReq" : Bool;   // PLC心跳
      "PLC.Unload_HeartbeatSignal" : Bool;
   END_VAR
BEGIN
END_DATA_BLOCK

DATA_BLOCK "Scanner1LoadData"   // DB530
{ S7_Optimized_Access := 'FALSE' }
// stored: AutoNumber false
   VAR
      "PLC.Station1DMXCode" : Int;
      "PLC.Station1RecipeNo" : Int;
      "PLC.PartTypeID" : String[128];
      Spare : Byte;
      "MES.ErrorCode" : Int;
      "MES.StatusBits" : DInt;
      "MES.Cycle_ID" : DInt;
      "MES.Unit_ParttypeID" : Int;
   END_VAR
BEGIN
END_DATA_BLOCK

DATA_BLOCK "Station1LoadData"   // DB510
{ S7_Optimized_Access := 'FALSE' }
// stored: AutoNumber false
   VAR
      "PLC.PartTypeID" : Int;
      "PLC.Station1RecipeNo" : Int;
      "PLC.Station1DMXCode" : String[128];
      "PLC.StationStatus" : Int;
      "MES.ErrorCode" : Int;
      "MES.StatusBits" : DInt;
      "MES.Cycle_ID" : DInt;
      "MES.Unit_ParttypeID" : Int;
   END_VAR
BEGIN
END_DATA_BLOCK

DATA_BLOCK "Station1UnLoadData"   // DB511
{ S7_Optimized_Access := 'FALSE' }
// stored: AutoNumber false
   VAR
      "PLC.PartTypeID" : Int;
      "PLC.Station1DMXCode" : String[128];
      "PLC.Station1RecipeNo" : Int;
      "PLC.PartStatus" : Int;
      "PLC.SubPartSN1" : String[128];
      "PLC.TransferTime" : String[128];
      Spare : Byte;
      Spare_1 : Byte;
      Spare_2 : Byte;
      Spare_3 : Byte;
      Spare_4 : Byte;
      Spare_5 : Byte;
      Spare_6 : Byte;
      Spare_7 : Byte;
      Spare_8 : Byte;
      Spare_9 : Byte;
      Spare_10 : Byte;
      "MES.ErrorCode" : Int;
      "MES.ErrorMsg" : String[128];
   END_VAR
BEGIN
END_DATA_BLOCK

DATA_BLOCK "Station2LoadData"   // DB512
{ S7_Optimized_Access := 'FALSE' }
// stored: AutoNumber false
   VAR
      "PLC.PartTypeID" : Int;
      "PLC.Station2RecipeNo" : Int;
      "PLC.Station2DMXCode" : String[128];
      "PLC.SubPartSN1" : String[128];
      "MES.ErrorCode" : Int;
      "MES.StatusBits" : DInt;
      "MES.Cycle_ID" : DInt;
      "MES.Unit_ParttypeID" : Int;
   END_VAR
BEGIN
END_DATA_BLOCK

DATA_BLOCK "Station2UnLoadData"   // DB513
{ S7_Optimized_Access := 'FALSE' }
// stored: AutoNumber false
   VAR
      "PLC.PartTypeID" : Int;
      "PLC.Station2DMXCode" : String[128];
      "PLC.Station2RecipeNo" : Int;
      "PLC.PartStatus" : Int;
      "PLC.SubPartSN1" : String[128];
      "PLC.TransferTime" : String[128];
      Spare : Byte;
      Spare_1 : Byte;
      Spare_2 : Byte;
      Spare_3 : Byte;
      Spare_4 : Byte;
      Spare_5 : Byte;
      Spare_6 : Byte;
      Spare_7 : Byte;
      Spare_8 : Byte;
      Spare_9 : Byte;
      Spare_10 : Byte;
      "MES.ErrorCode" : Int;
      "MES.ErrorMsg" : String[128];
   END_VAR
BEGIN
END_DATA_BLOCK

DATA_BLOCK "Station3LoadData"   // DB514
{ S7_Optimized_Access := 'FALSE' }
// stored: AutoNumber false
   VAR
      "PLC.PartTypeID" : Int;
      "PLC.Station3RecipeNo" : Int;
      "PLC.Station3DMXCode" : String[128];
      "PLC.SubPartSN1" : String[128];
      "MES.ErrorCode" : Int;
      "MES.StatusBits" : DInt;
      "MES.Cycle_ID" : DInt;
      "MES.Unit_ParttypeID" : Int;
   END_VAR
BEGIN
END_DATA_BLOCK

DATA_BLOCK "Station3UnLoadData"   // DB515
{ S7_Optimized_Access := 'FALSE' }
// stored: AutoNumber false
   VAR
      "PLC.PartTypeID" : Int;
      "PLC.Station3DMXCode" : String[50];
      "PLC.Station3RecipeNo" : Int;
      "PLC.PartStatus" : Int;
      "PLC.SubPartSN1" : String[50];
      "PLC.TransferTime" : String[50];
      "PLC.Power" : Real;
      "PLC.Displacement" : Real;
      "PLC.Program" : Int;
      "PLC.NGCode" : Int;
      Spare_2 : Byte;
      Spare_3 : Byte;
      Spare_4 : Byte;
      Spare_5 : Byte;
      Spare_6 : Byte;
      Spare_7 : Byte;
      Spare_8 : Byte;
      "MES.ErrorCode" : Int;
      Static_1 : String[60];
   END_VAR
BEGIN
END_DATA_BLOCK

DATA_BLOCK "Station4LoadData"   // DB516
{ S7_Optimized_Access := 'FALSE' }
// stored: AutoNumber false
   VAR
      "PLC.PartTypeID" : Int;
      "PLC.Station4RecipeNo" : Int;
      "PLC.Station4DMXCode" : String[128];
      "PLC.SubPartSN1" : String[128];
      "MES.ErrorCode" : Int;
      "MES.StatusBits" : DInt;
      "MES.Cycle_ID" : DInt;
      "MES.Unit_ParttypeID" : Int;
   END_VAR
BEGIN
END_DATA_BLOCK

DATA_BLOCK "Station4UnLoadData"   // DB517
{ S7_Optimized_Access := 'FALSE' }
// stored: AutoNumber false
   VAR
      "PLC.PartTypeID" : Int;
      "PLC.Station4DMXCode" : String[50];
      "PLC.Station4RecipeNo" : Int;
      "PLC.PartStatus" : Int;
      "PLC.SubPartSN1" : String[50];
      "PLC.TransferTime" : String[50];
      Spare : Byte;
      Spare_1 : Byte;
      Spare_2 : Byte;
      Spare_3 : Byte;
      Spare_4 : Byte;
      Spare_5 : Byte;
      Spare_6 : Byte;
      Spare_7 : Byte;
      Spare_8 : Byte;
      Spare_9 : Byte;
      Spare_10 : Byte;
      "MES.ErrorCode" : Int;
      "MES.ErrorMsg" : String[60];
   END_VAR
BEGIN
END_DATA_BLOCK

DATA_BLOCK "Station5LoadData"   // DB518
{ S7_Optimized_Access := 'FALSE' }
// stored: AutoNumber false
   VAR
      "PLC.PartTypeID" : Int;
      "PLC.Station5RecipeNo" : Int;
      "PLC.Station5DMXCode" : String[128];
      "PLC.SubPartSN1" : String[128];
      "MES.ErrorCode" : Int;
      "MES.StatusBits" : DInt;
      "MES.Cycle_ID" : DInt;
      "MES.Unit_ParttypeID" : Int;
   END_VAR
BEGIN
END_DATA_BLOCK

DATA_BLOCK "Station5UnLoadData"   // DB519
{ S7_Optimized_Access := 'FALSE' }
// stored: AutoNumber false
   VAR
      "PLC.PartTypeID" : Int;
      "PLC.Station5DMXCode" : String[50];
      "PLC.Station5RecipeNo" : Int;
      "PLC.PartStatus" : Int;
      "PLC.SubPartSN1" : String[50];
      "PLC.TransferTime" : String[50];
      "PLC.ShaftGlueIVPro" : Int;
      "PLC.ShaftGlueResult" : Int;
      "PLC.ShaftGlueIVScore1" : Int;
      "PLC.ShaftGlueIVScore2" : Int;
      "PLC.ShaftGlueIVScore3" : Int;
      "PLC.ShaftGlueIVScore4" : Int;
      "PLC.ShaftMagnetIVPro" : Int;
      "PLC.MagnetGlueResult" : Int;
      "PLC.MagnetIVScore" : Int;
      "PLC.GluePro" : Int;
      "PLC.NGCode" : Int;
      Spare_5 : Int;
      Spare_6 : Int;
      Spare_7 : Int;
      Spare_8 : Int;
      Spare_9 : Int;
      Spare_10 : Int;
      "MES.ErrorCode" : Int;
      "MES.ErrorMsg" : String[60];
   END_VAR
BEGIN
END_DATA_BLOCK

DATA_BLOCK "Station6LoadData"   // DB520
{ S7_Optimized_Access := 'FALSE' }
// stored: AutoNumber false
   VAR
      "PLC.PartTypeID" : Int;
      "PLC.Station6RecipeNo" : Int;
      "PLC.Station6DMXCode" : String[128];
      "PLC.SubPartSN1" : String[128];
      "MES.ErrorCode" : Int;
      "MES.StatusBits" : DInt;
      "MES.Cycle_ID" : DInt;
      "MES.Unit_ParttypeID" : Int;
   END_VAR
BEGIN
END_DATA_BLOCK

DATA_BLOCK "Station6UnLoadData"   // DB521
{ S7_Optimized_Access := 'FALSE' }
// stored: AutoNumber false
   VAR
      "PLC.PartTypeID" : Int;
      "PLC.Station6DMXCode" : String[50];
      "PLC.Station6RecipeNo" : Int;
      "PLC.PartStatus" : Int;
      "PLC.SubPartSN1" : String[50];
      "PLC.TransferTime" : String[50];
      Spare : Byte;
      Spare_1 : Byte;
      Spare_2 : Byte;
      Spare_3 : Byte;
      Spare_4 : Byte;
      Spare_5 : Byte;
      Spare_6 : Byte;
      Spare_7 : Byte;
      Spare_8 : Byte;
      Spare_9 : Byte;
      Spare_10 : Byte;
      "MES.ErrorCode" : Int;
      "MES.ErrorMsg" : String[60];
   END_VAR
BEGIN
END_DATA_BLOCK

DATA_BLOCK "Station7LoadData"   // DB522
{ S7_Optimized_Access := 'FALSE' }
// stored: AutoNumber false
   VAR
      "PLC.PartTypeID" : Int;
      "PLC.Station7RecipeNo" : Int;
      "PLC.Station7DMXCode" : String[128];
      "PLC.SubPartSN1" : String[128];
      "MES.ErrorCode" : Int;
      "MES.StatusBits" : DInt;
      "MES.Cycle_ID" : DInt;
      "MES.Unit_ParttypeID" : Int;
   END_VAR
BEGIN
END_DATA_BLOCK

DATA_BLOCK "Station7UnLoadData"   // DB523
{ S7_Optimized_Access := 'FALSE' }
// stored: AutoNumber false
   VAR
      "PLC.PartTypeID" : Int;
      "PLC.Station7DMXCode" : String[50];
      "PLC.Station7RecipeNo" : Int;
      "PLC.PartStatus" : Int;
      "PLC.SubPartSN1" : String[50];
      "PLC.TransferTime" : String[50];
      "PLC.Power" : Real;
      "PLC.Displacement" : Real;
      "PLC.Program" : Int;
      "PLC.NGCode" : Int;
      Spare_2 : Byte;
      Spare_3 : Byte;
      Spare_4 : Byte;
      Spare_5 : Byte;
      Spare_6 : Byte;
      Spare_7 : Byte;
      Spare_8 : Byte;
      "MES.ErrorCode" : Int;
      "MES.ErrorMsg" : String[60];
   END_VAR
BEGIN
END_DATA_BLOCK

DATA_BLOCK "Station8LoadData"   // DB524
{ S7_Optimized_Access := 'FALSE' }
// stored: AutoNumber false
   VAR
      "PLC.PartTypeID" : Int;
      "PLC.Station8RecipeNo" : Int;
      "PLC.Station8DMXCode" : String[128];
      Spare : Byte;
      "MES.ErrorCode" : Int;
      "MES.StatusBits" : DInt;
      "MES.Cycle_ID" : DInt;
      "MES.Unit_ParttypeID" : Int;
   END_VAR
BEGIN
END_DATA_BLOCK

DATA_BLOCK "Station8UnLoadData"   // DB525
{ S7_Optimized_Access := 'FALSE' }
// stored: AutoNumber false
   VAR
      "PLC.PartTypeID" : Int;
      "PLC.Station7DMXCode" : String[50];
      "PLC.Station7RecipeNo" : Int;
      "PLC.PartStatus" : Int;
      "PLC.SubPartSN1" : String[50];
      "PLC.TransferTime" : String[50];
      "PLC.Power" : Real;
      "PLC.Displacement" : Real;
      Spare : Byte;
      Spare_1 : Byte;
      Spare_2 : Byte;
      Spare_3 : Byte;
      Spare_4 : Byte;
      Spare_5 : Byte;
      Spare_6 : Byte;
      Spare_7 : Byte;
      Spare_8 : Byte;
      "MES.ErrorCode" : Int;
      "MES.ErrorMsg" : String[60];
   END_VAR
BEGIN
END_DATA_BLOCK

DATA_BLOCK "PartData_Interface_DB"   // DB1500
{ S7_Optimized_Access := 'TRUE' }
// stored: MemoryReserve 100
   VAR
      PartDataID : Int := 1;   // 物料数据序号
      PartData { S7_SetPoint := 'True'} : Array[1..4] of "PartData_UDT";
      PartCMD : Array[1..4] of Struct
         Set : Bool;
         Use : Bool;
      END_STRUCT;
   END_VAR
BEGIN
   // PartData[1] : XXX物料
   // PartData[2] : XXX物料
   // PartData[3] : XXX物料
   // PartData[4] : XXX物料
END_DATA_BLOCK

DATA_BLOCK "ChangeOver_DB"   // DB1700
{ S7_Optimized_Access := 'FALSE' }
// stored: AutoNumber false
   VAR RETAIN
      Robot_1 : Struct
         Req_RobotToMaintenancePos : Bool;
         Req_RobotToHomePos : Bool;
         Sensor_3 : Bool;
         Sensor_4 : Bool;
         Sensor_5 : Bool;
         Sensor_6 : Bool;
         Sensor_7 : Bool;
         Sensor_8 : Bool;
         EmptyProcess : Bool;
         EmptyFinish : Bool;
         Spare : Bool;
         HMI_MaintenancePosReqSel : Bool;
         HMI_MaintenancePosActive : Bool;
         MaintenancePosReqSelFlag : Bool;
         HMI_MaintenanceHomeReq : Bool;
         NoTaskRunning : Bool;
         Spare_6 : Bool;
         "Step" : Int;
      END_STRUCT;
      Robot_2 : Struct
         Req_RobotToMaintenancePos : Bool;
         Req_RobotToHomePos : Bool;
         Sensor_3 : Bool;
         Sensor_4 : Bool;
         Sensor_5 : Bool;
         Sensor_6 : Bool;
         Sensor_7 : Bool;
         Sensor_8 : Bool;
         EmptyProcess : Bool;
         EmptyFinish : Bool;
         Spare : Bool;
         HMI_MaintenancePosReqSel : Bool;
         HMI_MaintenancePosActive : Bool;
         MaintenancePosReqSelFlag : Bool;
         HMI_MaintenanceHomeReq : Bool;
         NoTaskRunning : Bool;
         Spare_6 : Bool;
         "Step" : Int;
      END_STRUCT;
      Robot_3 : Struct
         Req_RobotToMaintenancePos : Bool;
         Req_RobotToHomePos : Bool;
         Sensor_3 : Bool;
         Sensor_4 : Bool;
         Sensor_5 : Bool;
         Sensor_6 : Bool;
         Sensor_7 : Bool;
         Sensor_8 : Bool;
         EmptyProcess : Bool;
         EmptyFinish : Bool;
         Spare : Bool;
         HMI_MaintenancePosReqSel : Bool;
         HMI_MaintenancePosActive : Bool;
         MaintenancePosReqSelFlag : Bool;
         HMI_MaintenanceHomeReq : Bool;
         NoTaskRunning : Bool;
         Spare_6 : Bool;
         "Step" : Int;
      END_STRUCT;
      H_Line : Struct
         Sensor_1 : Bool;
         Sensor_2 : Bool;
         Sensor_3 : Bool;
         Sensor_4 : Bool;
         Sensor_5 : Bool;
         Sensor_6 : Bool;
         Sensor_7 : Bool;
         Sensor_8 : Bool;
         Sensor_9 : Bool;
         Sensor_10 : Bool;
         Sensor_11 : Bool;
         Sensor_12 : Bool;
         Sensor_13 : Bool;
         Sensor_14 : Bool;
         Sensor_15 : Bool;
         Sensor_16 : Bool;
         EmptyProcess : Bool;
         EmptyFinish : Bool;
         Spare : Bool;
         Spare_1 : Bool;
         Spare_2 : Bool;
         Spare_3 : Bool;
         Spare_4 : Bool;
         Spare_5 : Bool;
         Spare_6 : Bool;
         "Step" : Int;
      END_STRUCT;
      J_Line : Struct
         Sensor_1 : Bool;
         Sensor_2 : Bool;
         Sensor_3 : Bool;
         Sensor_4 : Bool;
         Sensor_5 : Bool;
         Sensor_6 : Bool;
         Sensor_7 : Bool;
         Sensor_8 : Bool;
         Sensor_9 : Bool;
         Sensor_10 : Bool;
         Sensor_11 : Bool;
         Sensor_12 : Bool;
         Sensor_13 : Bool;
         Sensor_14 : Bool;
         Sensor_15 : Bool;
         Sensor_16 : Bool;
         EmptyProcess : Bool;
         EmptyFinish : Bool;
         Spare : Bool;
         Spare_1 : Bool;
         Spare_2 : Bool;
         Spare_3 : Bool;
         Spare_4 : Bool;
         Spare_5 : Bool;
         Spare_6 : Bool;
         "Step" : Int;
      END_STRUCT;
      K_Line : Struct
         Sensor_1 : Bool;
         Sensor_2 : Bool;
         Sensor_3 : Bool;
         Sensor_4 : Bool;
         Sensor_5 : Bool;
         Sensor_6 : Bool;
         Sensor_7 : Bool;
         Sensor_8 : Bool;
         Sensor_9 : Bool;
         Sensor_10 : Bool;
         Sensor_11 : Bool;
         Sensor_12 : Bool;
         Sensor_13 : Bool;
         Sensor_14 : Bool;
         Sensor_15 : Bool;
         Sensor_16 : Bool;
         EmptyProcess : Bool;
         EmptyFinish : Bool;
         Spare : Bool;
         Spare_1 : Bool;
         Spare_2 : Bool;
         Spare_3 : Bool;
         Spare_4 : Bool;
         Spare_5 : Bool;
         Spare_6 : Bool;
         "Step" : Int;
      END_STRUCT;
      L_Line : Struct
         Sensor_1 : Bool;
         Sensor_2 : Bool;
         Sensor_3 : Bool;
         Sensor_4 : Bool;
         Sensor_5 : Bool;
         Sensor_6 : Bool;
         Sensor_7 : Bool;
         Sensor_8 : Bool;
         Sensor_9 : Bool;
         Sensor_10 : Bool;
         Sensor_11 : Bool;
         Sensor_12 : Bool;
         Sensor_13 : Bool;
         Sensor_14 : Bool;
         Sensor_15 : Bool;
         Sensor_16 : Bool;
         EmptyProcess : Bool;
         EmptyFinish : Bool;
         Spare : Bool;
         Spare_1 : Bool;
         Spare_2 : Bool;
         Spare_3 : Bool;
         Spare_4 : Bool;
         Spare_5 : Bool;
         Spare_6 : Bool;
         "Step" : Int;
      END_STRUCT;
      Global : Struct
         AllFixtureScanCompareOk : Bool;
         ChangeOverRequest : Bool;
         ChangeOverToolScanFlag : Bool;
         ManualModeFlag : Bool;
         ScanFixtureFlag : Bool;
         Station_empty : Bool;
         ChangeOverSelected : Bool;
         ScanFixtureFlag_ChangeOver : Bool;
         A1_TableScanStart : Bool;
         A2_TableScanStart : Bool;
         Hmi_Confirm_ChangeOver : Bool;
         ChangeOverActive : Bool;
         Hmi_ForceChangeOver : Bool;
         Spare_13 : Bool;
         Spare_14 : Bool;
         Spare_15 : Bool;
      END_STRUCT;
      P : Array[0..20] of Bool;
      "Time" : Array[0..3] of TOF_TIME;
      Robot1 : Struct
         Ring1Weight : Int;
         ShaftWeight : Int;
         MagnetWeight : Int;
         Ring2Weight : Int;
      END_STRUCT;
      Robot2 : Struct
         Ring1Weight : Int;
         ShaftWeight : Int;
         MagnetWeight : Int;
         Ring2Weight : Int;
      END_STRUCT;
      Robot3 : Struct
         Ring1Weight : Int;
         ShaftWeight : Int;
         MagnetWeight : Int;
         Ring2Weight : Int;
      END_STRUCT;
   END_VAR
BEGIN
END_DATA_BLOCK

DATA_BLOCK "AutoProcess_HMI"   // DB1666
{ S7_Optimized_Access := 'TRUE' }
// stored: AutoNumber false, MemoryReserve 100
   VAR
      IndexProcess : Int;   // 1 A_ScanRotate, 2 F_Robot1Grip1, 3 F_Robot1Grip2, 4 B_Press1, 5 C_Glue, 6 F_Robot2Grip1, 7 F_Robot2Grip2, 8 C_GlueNGBuffer, 9 C_MagnScanNGBuffer, 10 B_Press2, 11 F_Robot3Grip1, 12 F_Robot3Grip2, 13 H_ShafeLine, 14 J_ShafeLine, 15 K_ShafeLine, 16 L_ShafeLine
      ActualSHowingData : "ProcessData";
      Data_handling : Struct
         DeleteData : Bool;
         UpdateData_switch : Bool;
         UpdateData_Confirm : Bool;   // 1. step - request to confirm old new data
         FinalConfirm_Write : Bool;   // 2. final acceptance for data update
         ChangePending : Bool;   // changes are ready for actual index
         ConfirmDialogActive : Bool;   // Confirm dialog active
         LastIndex : Int;   // internal - memory for last index
      END_STRUCT;
      StationHasProduct : Array[1..16] of Bool;
   END_VAR
BEGIN
END_DATA_BLOCK

DATA_BLOCK "ST10Cylinder"   // DB1020
{ S7_Optimized_Access := 'FALSE' }
// stored: AutoNumber false
   VAR RETAIN
      Cy { S7_SetPoint := 'True'} : Array[1..110] of "Cyl";
   END_VAR
BEGIN
   // Cy[1] : A-顶升模组-01阻挡气缸
   // Cy[2] : A-顶升模组-01升降气缸
   // Cy[3] : A-顶升模组-02阻挡气缸
   // Cy[4] : A-顶升模组-02升降气缸
   // Cy[5] : A-托盘缓存阻挡气缸
   // Cy[6] : C-贴标模组水平移动Y轴
   // Cy[7] : C-贴标模组垂直移动Z轴
   // Cy[8] : C-贴标模组螺标签切料真空吸附
   // Cy[9] : C-贴标模组标签取料真空吸附-02
   // Cy[10] : C-贴标模组换型气缸
   Cy[1..10].In.Error := false;
   Cy[1..10].In.GoWorkInterlock := false;
   Cy[1..10].In.GoHomeInterlock := false;
   Cy[1..10].In.WorkPositionSensor := false;
   Cy[1..10].In.HomePositionSensor := false;
   Cy[1].In.ValveType := false;
   Cy[2].In.ValveType := true;
   Cy[3].In.ValveType := false;
   Cy[4].In.ValveType := true;
   Cy[5].In.ValveType := false;
   Cy[6..10].In.ValveType := true;
   Cy[1..10].In.ManualOutputType := false;
   Cy[1..10].In.FaultTime := 50;
   Cy[1..10].In.OnPositionTime := 10;
   Cy[1..10].Inout.ManualGoWork := FALSE;
   Cy[1..10].Inout.ManualGoHome := FALSE;
   Cy[1..10].Inout.AutoGoWork := FALSE;
   Cy[1..10].Inout.AutoGoHome := FALSE;
   Cy[1..10].S.GoWorkTime := 0;
   Cy[1..10].S.GoHomeTime := 0;
   Cy[1..10].S.WorkFaultTime := 0;
   Cy[1..10].S.HomeFaultTime := 0;
   Cy[1..10].S.BothSensorOnTime := 0;
   Cy[1..10].S.Pulse100mSP := FALSE;
   Cy[1..10].S.AutoGoWorkP := FALSE;
   Cy[1..10].S.AutoGoHomeP := FALSE;
   Cy[1..10].S.GoWork100mSP := TRUE;
   Cy[1..10].S.GoHome100mSP := TRUE;
   Cy[1..10].S.BothSensorOn100mSP := TRUE;
   Cy[1..10].S.Alarm := FALSE;
   Cy[1..10].S.spare1 := FALSE;
   Cy[1..10].S.spare2 := 16#00;
   Cy[1..10].Out.GoWorkPosition := FALSE;
   Cy[1].Out.GoHomePosition := FALSE;
   Cy[2].Out.GoHomePosition := TRUE;
   Cy[3].Out.GoHomePosition := FALSE;
   Cy[4].Out.GoHomePosition := TRUE;
   Cy[5..10].Out.GoHomePosition := FALSE;
   Cy[1..9].Out.GoWPButtonActive := TRUE;
   Cy[10].Out.GoWPButtonActive := FALSE;
   Cy[1..9].Out.GoHPButtonActive := TRUE;
   Cy[10].Out.GoHPButtonActive := FALSE;
   Cy[1..10].Out.GoWorkFault := FALSE;
   Cy[1..10].Out.GoHomeFault := FALSE;
   Cy[1..10].Out.SensorPositionFault := FALSE;
   Cy[1].Out.CyNO := 16#01;
   Cy[2].Out.CyNO := 16#02;
   Cy[3].Out.CyNO := 16#03;
   Cy[4].Out.CyNO := 16#04;
   Cy[5].Out.CyNO := 16#05;
   Cy[6].Out.CyNO := 16#06;
   Cy[7].Out.CyNO := 16#07;
   Cy[8].Out.CyNO := 16#08;
   Cy[9].Out.CyNO := 16#09;
   Cy[10].Out.CyNO := 16#0A;
END_DATA_BLOCK

DATA_BLOCK "ST10_SafetyGate_InterfaceDB"   // DB1140
{ S7_Optimized_Access := 'TRUE' }
// stored: AutoNumber false, MemoryReserve 100
   VAR
      aDev { S7_SetPoint := 'True'} : Array[1..20] of "SafetyGateUDT";
      SafetyDoorLamp { S7_SetPoint := 'True'} : Array[1..20] of Bool;
      H : Struct
         Status_1 : Int;
         Status_2 : Int;
         Status_3 : Int;
         p : Array[0..20] of Bool;
      END_STRUCT;
      J : Struct
         Status_1 : Int;
         Status_2 : Int;
         Status_3 : Int;
         p : Array[0..20] of Bool;
      END_STRUCT;
      K : Struct
         Status_1 : Int;
         Status_2 : Int;
         Status_3 : Int;
         p : Array[0..20] of Bool;
      END_STRUCT;
      L : Struct
         Status_1 : Int;
         Status_2 : Int;
         Status_3 : Int;
         p : Array[0..20] of Bool;
      END_STRUCT;
   END_VAR
BEGIN
END_DATA_BLOCK

DATA_BLOCK "ST10_Stopper_InterfaceDB"   // DB1161
{ S7_Optimized_Access := 'TRUE' }
// stored: AutoNumber false, MemoryReserve 100
   VAR
      aDev { S7_SetPoint := 'True'} : Array[1..5] of "ST_Stopper";
      Command { S7_SetPoint := 'True'} : Array[1..5] of "UDT_Stopper_FB";
   END_VAR
BEGIN
END_DATA_BLOCK

DATA_BLOCK "OP10_GeneralAnalogDB"   // DB1080
{ S7_Optimized_Access := 'TRUE' }
// stored: AutoNumber false, MemoryReserve 0
   VAR RETAIN
      aDev : Array[1..2] of "ST_GeneralAnalog";
   END_VAR
BEGIN
END_DATA_BLOCK

DATA_BLOCK "ST10_PLC_GetDB"   // DB901
{ S7_Optimized_Access := 'FALSE' }
// stored: AutoNumber false
   VAR
      InData : Struct
         Global : Struct
            Beat : Bool;
            AutoRunning : Bool;
            Alarm : Bool;
            SystemStandby : Bool;
            AutoMode : Bool;
            ManualMode : Bool;
            Spare_4 : Bool;
            Spare_5 : Bool;
            Spare_6 : Bool;
            Spare_7 : Bool;
            Spare_8 : Bool;
            Spare_9 : Bool;
            Spare_10 : Bool;
            Spare_11 : Bool;
            Spare_12 : Bool;
            Spare_13 : Bool;
         END_STRUCT;
         Control : Struct
            AskPallet : Bool;
            PalletInPos : Bool;
            Spare_1 : Bool;
            Spare_2 : Bool;
            Spare_3 : Bool;
            Spare_4 : Bool;
            Spare_5 : Bool;
            Spare_6 : Bool;
            Spare_7 : Bool;
            Spare_8 : Bool;
            Spare_9 : Bool;
            Spare_10 : Bool;
            Spare_11 : Bool;
            Spare_12 : Bool;
            Spare_13 : Bool;
            Spare_14 : Byte;
            Spare_15 : Byte;
         END_STRUCT;
         Data : Struct
            CurrentTemperature_1 : Int;
            CurrentTemperature_2 : Int;
            SetTemperature : Int;
            SetSolidifyTime : Int;
            ActualSolidifyTime : Int;   // Min
            Spare_3 : Array[0..83] of Byte;
         END_STRUCT;
      END_STRUCT;
   END_VAR
BEGIN
END_DATA_BLOCK

DATA_BLOCK "ST10_PLC_PutDB"   // DB902
{ S7_Optimized_Access := 'FALSE' }
// stored: AutoNumber false
   VAR
      OutData : Struct
         Global : Struct
            Beat : Bool;
            AutoRunning : Bool;
            Alarm : Bool;
            Spare_1 : Bool;
            Spare_2 : Bool;
            Spare_3 : Bool;
            Spare_4 : Bool;
            Spare_5 : Bool;
            Spare_6 : Bool;
            Spare_7 : Bool;
            Spare_8 : Bool;
            Spare_9 : Bool;
            Spare_10 : Bool;
            Spare_11 : Bool;
            Spare_12 : Bool;
            Spare_13 : Bool;
         END_STRUCT;
         Control : Struct
            PalletOut : Bool;
            Spare_16 : Bool;
            Spare_1 : Bool;
            Spare_2 : Bool;
            Spare_3 : Bool;
            Spare_4 : Bool;
            Spare_5 : Bool;
            Spare_6 : Bool;
            Spare_7 : Bool;
            Spare_8 : Bool;
            Spare_9 : Bool;
            Spare_10 : Bool;
            Spare_11 : Bool;
            Spare_12 : Bool;
            Spare_13 : Bool;
            Spare_14 : Byte;
            Spare_15 : Byte;
         END_STRUCT;
         Data : Struct
            Spare_5 : Int;
            Spare_4 : Int;
            Spare_1 : Int;
            Spare_2 : Int;
            Spare_6 : Int;   // Min
            Spare_3 : Array[0..83] of Byte;
         END_STRUCT;
      END_STRUCT;
   END_VAR
BEGIN
END_DATA_BLOCK

DATA_BLOCK "DB_KeyenceCheckerIV3"   // DB2101
{ S7_Optimized_Access := 'TRUE' }
// stored: AutoNumber false, MemoryReserve 100
   VAR
      aDev { S7_SetPoint := 'True'} : Array[1..4] of "ST_KeyenceCheckerIV3";
   END_VAR
BEGIN
   aDev[1].Para.nInAdr1 := 465;
   aDev[2].Para.nInAdr1 := 435;
   aDev[1].Para.nInAdr2 := 466;
   aDev[2].Para.nInAdr2 := 434;
   aDev[1].Para.nInAdr3 := 467;
   aDev[2].Para.nInAdr3 := 433;
   aDev[1].Para.nInAdr4 := 468;
   aDev[2].Para.nInAdr4 := 432;
   aDev[1].Para.nInAdr5 := 354;
   aDev[2].Para.nInAdr5 := 431;
   aDev[1].Para.nInAdr6 := 469;
   aDev[2].Para.nInAdr6 := 430;
   aDev[1].Para.nInAdr7 := 470;
   aDev[2].Para.nInAdr7 := 429;
   aDev[1].Para.nInAdr8 := 471;
   aDev[2].Para.nInAdr8 := 428;
   aDev[1].Para.nInAdr9 := 472;
   aDev[2].Para.nInAdr9 := 427;
   aDev[1].Para.nInAdr10 := 473;
   aDev[2].Para.nInAdr10 := 426;
   aDev[1].Para.nInAdr11 := 474;
   aDev[2].Para.nInAdr11 := 425;
   aDev[1].Para.nInAdr12 := 475;
   aDev[2].Para.nInAdr12 := 424;
   aDev[1].Para.nInAdr13 := 476;
   aDev[2].Para.nInAdr13 := 423;
   aDev[1].Para.nInAdr14 := 477;
   aDev[2].Para.nInAdr14 := 422;
   aDev[1].Para.nInAdr15 := 478;
   aDev[2].Para.nInAdr15 := 421;
   aDev[1].Para.nInAdr16 := 479;
   aDev[2].Para.nInAdr16 := 420;
   aDev[1].Para.nInAdr17 := 480;
   aDev[2].Para.nInAdr17 := 419;
   aDev[1].Para.nInAdr18 := 481;
   aDev[2].Para.nInAdr18 := 418;
   aDev[1].Para.nInAdr19 := 482;
   aDev[2].Para.nInAdr19 := 417;
   aDev[1].Para.nInAdr20 := 483;
   aDev[2].Para.nInAdr20 := 416;
   aDev[1].Para.nInAdr21 := 484;
   aDev[2].Para.nInAdr21 := 415;
   aDev[1].Para.nInAdr22 := 485;
   aDev[2].Para.nInAdr22 := 414;
   aDev[1].Para.nInAdr23 := 486;
   aDev[2].Para.nInAdr23 := 413;
   aDev[1].Para.nInAdr24 := 487;
   aDev[2].Para.nInAdr24 := 412;
   aDev[1].Para.nInAdr25 := 488;
   aDev[2].Para.nInAdr25 := 411;
   aDev[1].Para.nInAdr26 := 489;
   aDev[2].Para.nInAdr26 := 410;
   aDev[1].Para.nInAdr27 := 509;
   aDev[2].Para.nInAdr27 := 409;
   aDev[1].Para.nInAdr28 := 510;
   aDev[2].Para.nInAdr28 := 408;
   aDev[1].Para.nInAdr29 := 511;
   aDev[2].Para.nInAdr29 := 407;
   aDev[1].Para.nInAdr30 := 512;
   aDev[2].Para.nInAdr30 := 406;
   aDev[1].Para.nInAdr31 := 513;
   aDev[2].Para.nInAdr31 := 405;
   aDev[1].Para.nInAdr32 := 514;
   aDev[2].Para.nInAdr32 := 404;
   aDev[1].Para.nInAdr33 := 515;
   aDev[2].Para.nInAdr33 := 403;
   aDev[1].Para.nInAdr34 := 516;
   aDev[2].Para.nInAdr34 := 402;
   aDev[1].Para.nInAdr35 := 517;
   aDev[2].Para.nInAdr35 := 401;
   aDev[1].Para.nInAdr36 := 518;
   aDev[2].Para.nInAdr36 := 400;
   aDev[1].Para.nInAdr37 := 519;
   aDev[2].Para.nInAdr37 := 399;
   aDev[1].Para.nInAdr38 := 520;
   aDev[2].Para.nInAdr38 := 398;
   aDev[1].Para.nInAdr39 := 521;
   aDev[2].Para.nInAdr39 := 397;
   aDev[1].Para.nInAdr40 := 522;
   aDev[2].Para.nInAdr40 := 396;
   aDev[1].Para.nInAdr41 := 523;
   aDev[2].Para.nInAdr41 := 395;
   aDev[1].Para.nInAdr42 := 524;
   aDev[2].Para.nInAdr42 := 394;
   aDev[1].Para.nInAdr43 := 525;
   aDev[2].Para.nInAdr43 := 393;
   aDev[1].Para.nInAdr44 := 526;
   aDev[2].Para.nInAdr44 := 392;
   aDev[1].Para.nInAdr45 := 527;
   aDev[2].Para.nInAdr45 := 391;
   aDev[1].Para.nInAdr46 := 528;
   aDev[2].Para.nInAdr46 := 390;
   aDev[1].Para.nInAdr47 := 529;
   aDev[2].Para.nInAdr47 := 389;
   aDev[1].Para.nInAdr48 := 530;
   aDev[2].Para.nInAdr48 := 388;
   aDev[1].Para.nInAdr49 := 531;
   aDev[2].Para.nInAdr49 := 387;
   aDev[1].Para.nInAdr50 := 532;
   aDev[2].Para.nInAdr50 := 386;
   aDev[1].Para.nInAdr51 := 533;
   aDev[2].Para.nInAdr51 := 385;
   aDev[1].Para.nInAdr52 := 534;
   aDev[2].Para.nInAdr52 := 384;
   aDev[1].Para.nInAdr53 := 535;
   aDev[2].Para.nInAdr53 := 383;
   aDev[1].Para.nInAdr54 := 536;
   aDev[2].Para.nInAdr54 := 382;
   aDev[1].Para.nInAdr55 := 373;
   aDev[2].Para.nInAdr55 := 381;
   aDev[1].Para.nInAdr56 := 537;
   aDev[2].Para.nInAdr56 := 380;
   aDev[1].Para.nInAdr57 := 377;
   aDev[2].Para.nInAdr57 := 379;
   aDev[1].Para.nInAdr58 := 538;
   aDev[2].Para.nInAdr58 := 376;
   aDev[1].Para.nInAdr59 := 539;
   aDev[2].Para.nInAdr59 := 375;
   aDev[1].Para.nInAdr60 := 540;
   aDev[2].Para.nInAdr60 := 374;
   aDev[1].Para.nInAdr61 := 541;
   aDev[2].Para.nInAdr61 := 372;
   aDev[1].Para.nInAdr62 := 542;
   aDev[2].Para.nInAdr62 := 371;
   aDev[1].Para.nInAdr63 := 543;
   aDev[2].Para.nInAdr63 := 370;
   aDev[1].Para.nInAdr64 := 544;
   aDev[2].Para.nInAdr64 := 369;
   aDev[1].Para.nInAdr65 := 545;
   aDev[2].Para.nInAdr65 := 368;
   aDev[1].Para.nInAdr66 := 546;
   aDev[2].Para.nInAdr66 := 367;
   aDev[1].Para.nInAdr67 := 547;
   aDev[2].Para.nInAdr67 := 366;
   aDev[1].Para.nInAdr68 := 548;
   aDev[2].Para.nInAdr68 := 365;
   aDev[1].Para.nInAdr69 := 549;
   aDev[2].Para.nInAdr69 := 364;
   aDev[1].Para.nInAdr70 := 550;
   aDev[2].Para.nInAdr70 := 363;
   aDev[1].Para.nOutAdr1 := 464;
   aDev[2].Para.nOutAdr1 := 436;
END_DATA_BLOCK

DATA_BLOCK "HMISystemDB"   // DB2201
{ S7_Optimized_Access := 'FALSE' }
// stored: AutoNumber false
   VAR RETAIN
      DisplayRows : Int;
      MaxPage : Int;
      Rows : Int;
      UnEnableGroup : Bool;
      DisplaySymbol : Bool;
      "DisplaySymbol Time" : Int;
      SymbolText : Array[1..4] of Int;
      HMICylinderBypass : Array[1..50] of Struct
         "BY" : Array[1..50] of Int;
      END_STRUCT;
      HMI_Axis : "HMI_Axis";
   END_VAR
BEGIN
   HMI_Axis.INPUT.Axis_ID := 1;
END_DATA_BLOCK

DATA_BLOCK "IAI_A1"   // DB2211
{ S7_Optimized_Access := 'FALSE' }
// stored: AutoNumber false
   VAR RETAIN
      In : Struct
         iInterlock : Bool;   // interlock
         "iManJog+" : Bool;   // positive motion/action/...manually
         "iManJog-" : Bool;   // negtive motion/action/...manually
         iAutoStart : Bool;   // negtive motion/action/...automaticly
         iHome : Bool;   // Homing
         iCancelTask : Bool;   // Cancel task
         iPauseTask : Bool;   // Pause task
         iManStart : Bool;   // positive motion/action/...automaticly
         iManListStart : Bool;
         iLimitSwitchActive : Bool := true;
         iLimitSoftActive : Bool := true;
         iRunningTimeout : Time;
         iHomingTimeout : Time;
         iAutoPosition : DInt;
         iAutoVelocity : Int;
         iManListPosition : DInt;
         iManListVelocity : Int;
         iManListNumber : Int;   // position list number
         iManPosition : DInt;
         iManVelocity : Int;
         iMode : Int;   // 1-相对;2-绝对
      END_STRUCT;
      Out : Struct
         oReady : Bool;
         oWarning : Bool;   // warning
         oError : Bool;   // error
         oInterlock : Bool;
         oServoEnable : Bool;
         oRunning : Bool;
         oHoming : Bool;
         oHomeRef : Bool;
         oServoPosOK : Bool;
         oErrorCode : Int;
         oStatus : Int;
         oActPosition : DInt;
         oManualListPos : DInt;
      END_STRUCT;
      IO : Struct
         ioManEnale : Bool;
         ioAutoEnale : Bool;
      END_STRUCT;
      Spare : Struct
         S : Array[0..100] of Byte;
      END_STRUCT;
      Manual : Struct
         Index : Int := 1;
         Pos : Array[1..20] of Struct
            Pos : Real;
            Vel : Int;
         END_STRUCT;
      END_STRUCT;
      Auto : Struct
         Index : Int := 1;
         Pos : Array[1..20] of Struct
            Pos : Real;
            Vel : Int;
         END_STRUCT;
      END_STRUCT;
      Interlock : Struct
         Active : Bool;
         Case1 : Bool;
         Case2 : Bool;
         Case3 : Bool;
         Case4 : Bool;
         Case5 : Bool;
         Case6 : Bool;
         Case7 : Bool;
         Case8 : Bool;
         Case9 : Bool;
         Case10 : Bool;
      END_STRUCT;
      PositionOk : Array[1..20] of Bool;
      Home_Pos : Struct
         "Home Pos Pls" : Bool;
         "Arrow indication" : Int;
         "Process prompt" : Int;
         "Button prompt" : Int;
      END_STRUCT;
   END_VAR
BEGIN
   // Auto.Pos[1] : 1.取料位置
   // Auto.Pos[2] : 2.放料位置
   // Auto.Pos[3] : 3.
   // Auto.Pos[4] : 4.
   // Auto.Pos[5] : 5.
   // Auto.Pos[6] : 6.
   // Auto.Pos[7] : 7.
   // Auto.Pos[8] : 8.
   // Auto.Pos[9] : 9.
   // PositionOk[1] : [1]
   // PositionOk[2] : [2]
   // PositionOk[3] : [3]
   // PositionOk[4] : [4]
   // PositionOk[5] : [5]
   // PositionOk[6] : [6]
   // PositionOk[7] : [7]
   // PositionOk[8] : [8]
   // PositionOk[9] : [9]
END_DATA_BLOCK

DATA_BLOCK "IAI_A2"   // DB2212
{ S7_Optimized_Access := 'FALSE' }
// stored: AutoNumber false
   VAR
      In : Struct
         iInterlock : Bool;   // interlock
         "iManJog+" : Bool;   // positive motion/action/...manually
         "iManJog-" : Bool;   // negtive motion/action/...manually
         iAutoStart : Bool;   // negtive motion/action/...automaticly
         iHome : Bool;   // Homing
         iCancelTask : Bool;   // Cancel task
         iPauseTask : Bool;   // Pause task
         iManStart : Bool;   // positive motion/action/...automaticly
         iManListStart : Bool;
         iLimitSwitchActive : Bool := true;
         iLimitSoftActive : Bool := true;
         iRunningTimeout : Time;
         iHomingTimeout : Time;
         iAutoPosition : DInt;
         iAutoVelocity : Int;
         iManListPosition : DInt;
         iManListVelocity : Int;
         iManListNumber : Int;   // position list number
         iManPosition : DInt;
         iManVelocity : Int;
         iMode : Int;   // 1-相对;2-绝对
      END_STRUCT;
      Out : Struct
         oReady : Bool;
         oWarning : Bool;   // warning
         oError : Bool;   // error
         oInterlock : Bool;
         oServoEnable : Bool;
         oRunning : Bool;
         oHoming : Bool;
         oHomeRef : Bool;
         oServoPosOK : Bool;
         oErrorCode : Int;
         oStatus : Int;
         oActPosition : DInt;
         oManualListPos : DInt;
      END_STRUCT;
      IO : Struct
         ioManEnale : Bool;
         ioAutoEnale : Bool;
      END_STRUCT;
      Spare : Struct
         S : Array[0..100] of Byte;
      END_STRUCT;
      Manual : Struct
         Index : Int := 1;
         Pos : Array[1..20] of Struct
            Pos : Real;
            Vel : Int;
         END_STRUCT;
      END_STRUCT;
      Auto : Struct
         Index : Int := 1;
         Pos : Array[1..20] of Struct
            Pos : Real;
            Vel : Int;
         END_STRUCT;
      END_STRUCT;
      Interlock : Struct
         Active : Bool;
         Case1 : Bool;
         Case2 : Bool;
         Case3 : Bool;
         Case4 : Bool;
         Case5 : Bool;
         Case6 : Bool;
         Case7 : Bool;
         Case8 : Bool;
         Case9 : Bool;
         Case10 : Bool;
      END_STRUCT;
      PositionOk : Array[1..20] of Bool;
      Home_Pos : Struct
         "Home Pos Pls" : Bool;
         "Arrow indication" : Int;
         "Process prompt" : Int;
         "Button prompt" : Int;
      END_STRUCT;
   END_VAR
BEGIN
   // Auto.Pos[1] : 1.取料位置
   // Auto.Pos[2] : 2.放料位置
   // Auto.Pos[3] : 3.
   // Auto.Pos[4] : 4.
   // Auto.Pos[5] : 5.
   // Auto.Pos[6] : 6.
   // Auto.Pos[7] : 7.
   // Auto.Pos[8] : 8.
   // Auto.Pos[9] : 9.
   // PositionOk[1] : [1]
   // PositionOk[2] : [2]
   // PositionOk[3] : [3]
   // PositionOk[4] : [4]
   // PositionOk[5] : [5]
   // PositionOk[6] : [6]
   // PositionOk[7] : [7]
   // PositionOk[8] : [8]
   // PositionOk[9] : [9]
END_DATA_BLOCK

DATA_BLOCK "IAI_A3"   // DB2213
{ S7_Optimized_Access := 'FALSE' }
// stored: AutoNumber false
   VAR
      In : Struct
         iInterlock : Bool;   // interlock
         "iManJog+" : Bool;   // positive motion/action/...manually
         "iManJog-" : Bool;   // negtive motion/action/...manually
         iAutoStart : Bool;   // negtive motion/action/...automaticly
         iHome : Bool;   // Homing
         iCancelTask : Bool;   // Cancel task
         iPauseTask : Bool;   // Pause task
         iManStart : Bool;   // positive motion/action/...automaticly
         iManListStart : Bool;
         iLimitSwitchActive : Bool := true;
         iLimitSoftActive : Bool := true;
         iRunningTimeout : Time;
         iHomingTimeout : Time;
         iAutoPosition : DInt;
         iAutoVelocity : Int;
         iManListPosition : DInt;
         iManListVelocity : Int;
         iManListNumber : Int;   // position list number
         iManPosition : DInt;
         iManVelocity : Int;
         iMode : Int;   // 1-相对;2-绝对
      END_STRUCT;
      Out : Struct
         oReady : Bool;
         oWarning : Bool;   // warning
         oError : Bool;   // error
         oInterlock : Bool;
         oServoEnable : Bool;
         oRunning : Bool;
         oHoming : Bool;
         oHomeRef : Bool;
         oServoPosOK : Bool;
         oErrorCode : Int;
         oStatus : Int;
         oActPosition : DInt;
         oManualListPos : DInt;
      END_STRUCT;
      IO : Struct
         ioManEnale : Bool;
         ioAutoEnale : Bool;
      END_STRUCT;
      Spare : Struct
         S : Array[0..100] of Byte;
      END_STRUCT;
      Manual : Struct
         Index : Int := 1;
         Pos : Array[1..20] of Struct
            Pos : Real;
            Vel : Int;
         END_STRUCT;
      END_STRUCT;
      Auto : Struct
         Index : Int := 1;
         Pos : Array[1..20] of Struct
            Pos : Real;
            Vel : Int;
         END_STRUCT;
      END_STRUCT;
      Interlock : Struct
         Active : Bool;
         Case1 : Bool;
         Case2 : Bool;
         Case3 : Bool;
         Case4 : Bool;
         Case5 : Bool;
         Case6 : Bool;
         Case7 : Bool;
         Case8 : Bool;
         Case9 : Bool;
         Case10 : Bool;
      END_STRUCT;
      PositionOk : Array[1..20] of Bool;
      Home_Pos : Struct
         "Home Pos Pls" : Bool;
         "Arrow indication" : Int;
         "Process prompt" : Int;
         "Button prompt" : Int;
      END_STRUCT;
   END_VAR
BEGIN
   // Auto.Pos[1] : 1.取料位置
   // Auto.Pos[2] : 2.放料位置
   // Auto.Pos[3] : 3.
   // Auto.Pos[4] : 4.
   // Auto.Pos[5] : 5.
   // Auto.Pos[6] : 6.
   // Auto.Pos[7] : 7.
   // Auto.Pos[8] : 8.
   // Auto.Pos[9] : 9.
   // PositionOk[1] : [1]
   // PositionOk[2] : [2]
   // PositionOk[3] : [3]
   // PositionOk[4] : [4]
   // PositionOk[5] : [5]
   // PositionOk[6] : [6]
   // PositionOk[7] : [7]
   // PositionOk[8] : [8]
   // PositionOk[9] : [9]
END_DATA_BLOCK

DATA_BLOCK "IAI_DeviceCtl"   // DB2204
{ S7_Optimized_Access := 'FALSE' }
// stored: AutoNumber false
   VAR RETAIN
      IAIServo : Array[1..4] of Struct
         i : Int;
         nError : Int;
         nWarning : Int;
         nPositionListNo : Int;
         Pos : "PosList_IAI";
         Point : Array[0..39] of Struct
            Start : Bool;
            Achieve : Bool;
         END_STRUCT;
      END_STRUCT;
   END_VAR
BEGIN
   IAIServo[1..4].nPositionListNo := 1;
   // IAIServo[1].Point[1] : 初始位 / 上料位1
   // IAIServo[1].Point[2] : 抓料位 / 上料位2
   // IAIServo[1].Point[3] : 上料拍照位 / 上料位3
   // IAIServo[1].Point[4] : 下料位1 / 上料位4
   // IAIServo[1].Point[5] : 下料位2 / 上料位5
   // IAIServo[1].Point[6] : 下料位3 / 上料位6
   // IAIServo[1].Point[7] : 下料位4 / 上料位7
   // IAIServo[1].Point[8] : 下料位5 / 上料位8
   // IAIServo[1].Point[9] : NG下料位
   // IAIServo[2].Point[1] : 初始位
   // IAIServo[2].Point[2] : 取料位1 / 扫码位置2
   // IAIServo[2].Point[3] : 取料位2 / 扫码位置3
   // IAIServo[2].Point[4] : 取料位3 / 扫码位置4
   // IAIServo[2].Point[5] : 取料位4 / 扫码位置5
   // IAIServo[2].Point[6] : 取料位5 / 扫码位置6
   // IAIServo[2].Point[7] : 清洁位 / 扫码位置7
   // IAIServo[2].Point[8] : NG位 / 扫码位置8
   // IAIServo[2].Point[9] : 快速装配位
   // IAIServo[2].Point[10] : 慢速装配位
END_DATA_BLOCK

DATA_BLOCK "ModeDB"   // DB2203
{ S7_Optimized_Access := 'FALSE' }
// stored: AutoNumber false
   VAR
      Gen { S7_SetPoint := 'True'} : "ModeGenStruct";
   END_VAR
BEGIN
END_DATA_BLOCK

DATA_BLOCK "ProcessData_1"   // DB2300
{ S7_Optimized_Access := 'FALSE' }
// stored: AutoNumber false
   VAR RETAIN
      AlwaysZero : Byte := 16#00;
      "OP40.2" : Struct
         Kistler_Continue_Interlock : Bool := FALSE;
         Kistler_Interlock : Bool := FALSE;
         KistlerPress_autoInterlock : Bool := FALSE;
         KistlerPress_1Flag : Bool := FALSE;
         KistlerPress_2Flag : Bool := FALSE;
         KistlerPress_1Flag_Reset : Bool := FALSE;
         KistlerPress_2Flag_Reset : Bool := FALSE;
         Spare_7 : Bool := FALSE;
         Spare_8 : Bool := FALSE;
         Spare_9 : Bool := FALSE;
         Spare_10 : Bool := FALSE;
         Spare_11 : Bool := FALSE;
         Spare_12 : Bool := FALSE;
         Spare_13 : Bool := FALSE;
         Spare_14 : Bool := FALSE;
         Spare_15 : Bool := FALSE;
      END_STRUCT;
      "OP40.3" : Struct
         Kistler_Continue_Interlock : Bool := FALSE;
         Kistler_Interlock : Bool := FALSE;
         KistlerPress_autoInterlock : Bool := FALSE;
         KistlerPress_1Flag : Bool := FALSE;
         KistlerPress_2Flag : Bool := FALSE;
         KistlerPress_1Flag_Reset : Bool := FALSE;
         KistlerPress_2Flag_Reset : Bool := FALSE;
         Spare_7 : Bool := FALSE;
         Spare_8 : Bool := FALSE;
         Spare_9 : Bool := FALSE;
         Spare_10 : Bool := FALSE;
         Spare_11 : Bool := FALSE;
         Spare_12 : Bool := FALSE;
         Spare_13 : Bool := FALSE;
         Spare_14 : Bool := FALSE;
         Spare_15 : Bool := FALSE;
      END_STRUCT;
      "HMI_OP40.2" { S7_SetPoint := 'True'} : "OP40_Data";
      "HMI_OP40.3" { S7_SetPoint := 'True'} : "OP40_Data";
      PressInterlock_1 { S7_SetPoint := 'True'} : Array[0..15] of Bool;
      PressInterlock_2 : Array[0..15] of Bool;
      Calibartion_1 : Bool;
      Calibartion_2 : Bool;
   END_VAR
BEGIN
   "HMI_OP40.2".AssemblyResult := 16#00;
   "HMI_OP40.2".SN := '';
   "HMI_OP40.2".ProcessData.AssemblyResult1 := 16#00;
   "HMI_OP40.2".ProcessData.AssemblyResult2 := 16#00;
   "HMI_OP40.2".ProcessData.StartForce1 := 0.0;
   "HMI_OP40.2".ProcessData.StartLVDT1 := 0.0;
   "HMI_OP40.2".ProcessData.ProcessForce1 := 0.0;
   "HMI_OP40.2".ProcessData.ProcessLVDT1 := 0.0;
   "HMI_OP40.2".ProcessData.EndForce1 := 0.0;
   "HMI_OP40.2".ProcessData.EndLVDT1 := 0.0;
   "HMI_OP40.2".ProcessData.StartForce2 := 0.0;
   "HMI_OP40.2".ProcessData.StartLVDT2 := 0.0;
   "HMI_OP40.2".ProcessData.ProcessForce2 := 0.0;
   "HMI_OP40.2".ProcessData.ProcessLVDT2 := 0.0;
   "HMI_OP40.2".ProcessData.EndForce2 := 0.0;
   "HMI_OP40.2".ProcessData.EndLVDT2 := 0.0;
   "HMI_OP40.3".AssemblyResult := 16#00;
   "HMI_OP40.3".SN := '';
   "HMI_OP40.3".ProcessData.AssemblyResult1 := 16#00;
   "HMI_OP40.3".ProcessData.AssemblyResult2 := 16#00;
   "HMI_OP40.3".ProcessData.StartForce1 := 0.0;
   "HMI_OP40.3".ProcessData.StartLVDT1 := 0.0;
   "HMI_OP40.3".ProcessData.ProcessForce1 := 0.0;
   "HMI_OP40.3".ProcessData.ProcessLVDT1 := 0.0;
   "HMI_OP40.3".ProcessData.EndForce1 := 0.0;
   "HMI_OP40.3".ProcessData.EndLVDT1 := 0.0;
   "HMI_OP40.3".ProcessData.StartForce2 := 0.0;
   "HMI_OP40.3".ProcessData.StartLVDT2 := 0.0;
   "HMI_OP40.3".ProcessData.ProcessForce2 := 0.0;
   "HMI_OP40.3".ProcessData.ProcessLVDT2 := 0.0;
   "HMI_OP40.3".ProcessData.EndForce2 := 0.0;
   "HMI_OP40.3".ProcessData.EndLVDT2 := 0.0;
END_DATA_BLOCK

DATA_BLOCK "Robot_DB"   // DB2405
{ S7_Optimized_Access := 'FALSE' }
// stored: AutoNumber false
   VAR
      LoadNG_1 : Array[1..5] of Bool;
      LoadNG_2 : Array[1..5] of Bool;
      LoadNG_3 : Array[1..5] of Bool;
      UnLoadNG_1 : Array[1..5] of Bool;
      UnLoadNG_2 : Array[1..5] of Bool;
      UnLoadNG_3 : Array[1..5] of Bool;
      P : Array[1..16] of Bool;
      RobotFlag_1 : Array[1..8] of Bool;
      RobotFlag_2 : Array[1..8] of Bool;
      RobotFlag_3 : Array[1..8] of Bool;
      RobotSpeed : Array[1..8] of USInt;
      TON : Array[1..18] of TON_TIME;
      Control : Struct
         Robot1GripControl : Bool;
         Robot2GripControl : Bool;
         Robot3GripControl : Bool;
      END_STRUCT;
      Robot_1 : Struct
         PalletCount_1 : Int;
         GripCompareCodeOK_1 : Bool;
         GripCompareCodeOK_2 : Bool;
         GripCompareCodeOK_3 : Bool;
         GripCompareCodeOK_4 : Bool;
         GripCompareCodeOK : Bool;
         Spare_8 : Bool;
         Spare_6 : Bool;
         Spare_7 : Bool;
         SpeedChangeFlag : Bool;
         MasteringTest_Req : Bool;
         BrakeTest_Req : Bool;
         Spare_11 : Bool;
         Spare_12 : Bool;
         Spare_13 : Bool;
         Spare_14 : Bool;
         Spare_15 : Bool;
         SpeedCount : Int;
      END_STRUCT;
      Robot_2 : Struct
         PalletCount_1 : Int;
         PalletCount_2 : Int;
         GripCompareCodeOK_1 : Bool;
         GripCompareCodeOK_2 : Bool;
         GripCompareCodeOK_3 : Bool;
         GripCompareCodeOK_4 : Bool;
         GripCompareCodeOK : Bool;
         Spare_5 : Bool;
         Spare_6 : Bool;
         Spare_7 : Bool;
         SpeedChangeFlag : Bool;
         MasteringTest_Req : Bool;
         BrakeTest_Req : Bool;
         Spare_11 : Bool;
         Spare_12 : Bool;
         Spare_13 : Bool;
         Spare_14 : Bool;
         Spare_15 : Bool;
         SpeedCount : Int;
      END_STRUCT;
      Robot_3 : Struct
         PalletCount_1 : Int;
         PalletCount_2 : Int;
         GripCompareCodeOK_1 : Bool;
         GripCompareCodeOK_2 : Bool;
         GripCompareCodeOK_3 : Bool;
         GripCompareCodeOK_4 : Bool;
         GripCompareCodeOK : Bool;
         Spare_5 : Bool;
         Spare_6 : Bool;
         Spare_7 : Bool;
         SpeedChangeFlag : Bool;
         MasteringTest_Req : Bool;
         BrakeTest_Req : Bool;
         Spare_11 : Bool;
         Spare_12 : Bool;
         Spare_13 : Bool;
         Spare_14 : Bool;
         Spare_15 : Bool;
         SpeedCount : Int;
      END_STRUCT;
   END_VAR
BEGIN
END_DATA_BLOCK

DATA_BLOCK "Debug"   // DB5
{ S7_Optimized_Access := 'TRUE' }
// stored: AutoNumber false, MemoryReserve 100
   VAR
      Bypass : Array[0..100] of Bool;
      Squence : Array[0..100] of Bool;
   END_VAR
BEGIN
   Bypass[3] := 0;
END_DATA_BLOCK

DATA_BLOCK "ServoV90_A1"   // DB2501
{ S7_Optimized_Access := 'FALSE' }
// stored: AutoNumber false
   VAR RETAIN
      In : Struct
         iInterlock : Bool := TRUE;   // interlock
         "iManJog+" : Bool := FALSE;   // positive motion/action/...manually
         "iManJog-" : Bool := FALSE;   // negtive motion/action/...manually
         iAutoStart : Bool := FALSE;   // negtive motion/action/...automaticly
         iHome : Bool := FALSE;   // Homing
         iCancelTask : Bool := FALSE;   // Cancel task
         iPauseTask : Bool := FALSE;   // Pause task
         iManStart : Bool := FALSE;   // positive motion/action/...automaticly
         iManListStart : Bool := FALSE;
         iLimitSwitchActive : Bool := TRUE;
         iLimitSoftActive : Bool := TRUE;
         iRunningTimeout : Time := T#0MS;
         iHomingTimeout : Time := T#0MS;
         iAutoPosition : DInt := 0;
         iAutoVelocity : Int := 0;
         iManListPosition : DInt := 0;
         iManListVelocity : Int := 10000;
         iManListNumber : Int := 0;   // position list number
         iManPosition : DInt := 318250;
         iManVelocity : Int := 10000;
         iMode : Int := 0;   // 1-相对;2-绝对
      END_STRUCT;
      Out : Struct
         oReady : Bool := FALSE;
         oWarning : Bool := FALSE;   // warning
         oError : Bool := TRUE;   // error
         oInterlock : Bool := TRUE;
         oServoEnable : Bool := FALSE;
         oRunning : Bool := FALSE;
         oHoming : Bool := FALSE;
         oHomeRef : Bool := TRUE;
         oServoPosOK : Bool := FALSE;
         oErrorCode : Int := -244;
         oStatus : Int := 0;
         oActPosition : DInt := 93294;
         oManualListPos : DInt := 3419;
      END_STRUCT;
      IO : Struct
         ioManEnale : Bool := FALSE;
         ioAutoEnale : Bool := FALSE;
      END_STRUCT;
      Spare : Struct
         S : Array[0..100] of Byte;
      END_STRUCT;
      Manual : Struct
         Index : Int := 1;
         Pos : Array[1..20] of Struct
            Pos : DInt;
            Vel : Int;
         END_STRUCT;
      END_STRUCT;
      Auto : Struct
         Index : Int := 6;
         Pos : Array[1..20] of Struct
            Pos : DInt;
            Vel : Int;
         END_STRUCT;
      END_STRUCT;
      Interlock : Struct
         Active : Bool := FALSE;
         Case1 : Bool := TRUE;
         Case2 : Bool := TRUE;
         Case3 : Bool := FALSE;
         Case4 : Bool := FALSE;
         Case5 : Bool := FALSE;
         Case6 : Bool := FALSE;
         Case7 : Bool := FALSE;
         Case8 : Bool := FALSE;
         Case9 : Bool := FALSE;
         Case10 : Bool := FALSE;
      END_STRUCT;
      PositionOk : Array[1..20] of Bool;
      Home_Pos : Struct
         "Home Pos Pls" : Bool := FALSE;
         "Arrow indication" : Int := 0;
         "Process prompt" : Int := 0;
         "Button prompt" : Int := 0;
      END_STRUCT;
   END_VAR
BEGIN
   Spare.S[0..100] := 16#00;
   Manual.Pos[1].Pos := 3419;
   Manual.Pos[2].Pos := 48386;
   Manual.Pos[3].Pos := 93294;
   Manual.Pos[4].Pos := 138335;
   Manual.Pos[5].Pos := 183464;
   Manual.Pos[6].Pos := 228443;
   Manual.Pos[7].Pos := 273535;
   Manual.Pos[8].Pos := 318250;
   Manual.Pos[9..20].Pos := 0;
   Manual.Pos[1..8].Vel := 10000;
   Manual.Pos[9..20].Vel := 0;
   Auto.Pos[1].Pos := 3419;
   Auto.Pos[2].Pos := 48386;
   Auto.Pos[3].Pos := 93294;
   Auto.Pos[4].Pos := 138335;
   Auto.Pos[5].Pos := 183464;
   Auto.Pos[6].Pos := 228443;
   Auto.Pos[7].Pos := 273535;
   Auto.Pos[8].Pos := 318250;
   Auto.Pos[9..20].Pos := 0;
   Auto.Pos[1..8].Vel := 10000;
   Auto.Pos[9..20].Vel := 0;
   // Auto.Pos[1] : 1.取料位置
   // Auto.Pos[2] : 2.放料位置
   // Auto.Pos[3] : 3.
   // Auto.Pos[4] : 4.
   // Auto.Pos[5] : 5.
   // Auto.Pos[6] : 6.
   // Auto.Pos[7] : 7.
   // Auto.Pos[8] : 8.
   // Auto.Pos[9] : 9.
   PositionOk[1] := FALSE;   // [1]
   PositionOk[2] := FALSE;   // [2]
   PositionOk[3] := FALSE;   // [3]
   PositionOk[4] := FALSE;   // [4]
   PositionOk[5] := FALSE;   // [5]
   PositionOk[6] := FALSE;   // [6]
   PositionOk[7] := FALSE;   // [7]
   PositionOk[8] := FALSE;   // [8]
   PositionOk[9] := FALSE;   // [9]
   PositionOk[10..20] := FALSE;
END_DATA_BLOCK

DATA_BLOCK "ServoV90_A2"   // DB2502
{ S7_Optimized_Access := 'FALSE' }
// stored: AutoNumber false
   VAR
      In : Struct
         iInterlock : Bool := TRUE;   // interlock
         "iManJog+" : Bool := FALSE;   // positive motion/action/...manually
         "iManJog-" : Bool := FALSE;   // negtive motion/action/...manually
         iAutoStart : Bool := FALSE;   // negtive motion/action/...automaticly
         iHome : Bool := FALSE;   // Homing
         iCancelTask : Bool := FALSE;   // Cancel task
         iPauseTask : Bool := FALSE;   // Pause task
         iManStart : Bool := FALSE;   // positive motion/action/...automaticly
         iManListStart : Bool := FALSE;
         iLimitSwitchActive : Bool := TRUE;
         iLimitSoftActive : Bool := TRUE;
         iRunningTimeout : Time := T#0MS;
         iHomingTimeout : Time := T#0MS;
         iAutoPosition : DInt := 0;
         iAutoVelocity : Int := 0;
         iManListPosition : DInt := 0;
         iManListVelocity : Int := 0;
         iManListNumber : Int := 0;   // position list number
         iManPosition : DInt := 0;
         iManVelocity : Int := 0;
         iMode : Int := 0;   // 1-相对;2-绝对
      END_STRUCT;
      Out : Struct
         oReady : Bool := FALSE;
         oWarning : Bool := FALSE;   // warning
         oError : Bool := TRUE;   // error
         oInterlock : Bool := TRUE;
         oServoEnable : Bool := FALSE;
         oRunning : Bool := FALSE;
         oHoming : Bool := FALSE;
         oHomeRef : Bool := TRUE;
         oServoPosOK : Bool := FALSE;
         oErrorCode : Int := -244;
         oStatus : Int := 0;
         oActPosition : DInt := 113;
         oManualListPos : DInt := 0;
      END_STRUCT;
      IO : Struct
         ioManEnale : Bool := FALSE;
         ioAutoEnale : Bool := FALSE;
      END_STRUCT;
      Spare : Struct
         S : Array[0..100] of Byte;
      END_STRUCT;
      Manual : Struct
         Index : Int := 1;
         Pos : Array[1..20] of Struct
            Pos : DInt;
            Vel : Int;
         END_STRUCT;
      END_STRUCT;
      Auto : Struct
         Index : Int := 1;
         Pos : Array[1..20] of Struct
            Pos : DInt;
            Vel : Int;
         END_STRUCT;
      END_STRUCT;
      Interlock : Struct
         Active : Bool := FALSE;
         Case1 : Bool := TRUE;
         Case2 : Bool := TRUE;
         Case3 : Bool := FALSE;
         Case4 : Bool := FALSE;
         Case5 : Bool := FALSE;
         Case6 : Bool := FALSE;
         Case7 : Bool := FALSE;
         Case8 : Bool := FALSE;
         Case9 : Bool := FALSE;
         Case10 : Bool := FALSE;
      END_STRUCT;
      PositionOk : Array[1..20] of Bool;
      Home_Pos : Struct
         "Home Pos Pls" : Bool := FALSE;
         "Arrow indication" : Int := 0;
         "Process prompt" : Int := 0;
         "Button prompt" : Int := 0;
      END_STRUCT;
   END_VAR
BEGIN
   Spare.S[0..100] := 16#00;
   Manual.Pos[1].Pos := 0;
   Manual.Pos[2].Pos := 450000;
   Manual.Pos[3].Pos := 900000;
   Manual.Pos[4].Pos := 135000;
   Manual.Pos[5].Pos := 180000;
   Manual.Pos[6].Pos := 225000;
   Manual.Pos[7].Pos := 270000;
   Manual.Pos[8].Pos := 315000;
   Manual.Pos[9..20].Pos := 0;
   Manual.Pos[1..8].Vel := 10000;
   Manual.Pos[9..20].Vel := 0;
   Auto.Pos[1].Pos := 0;
   Auto.Pos[2].Pos := 450000;
   Auto.Pos[3].Pos := 900000;
   Auto.Pos[4].Pos := 135000;
   Auto.Pos[5].Pos := 180000;
   Auto.Pos[6].Pos := 225000;
   Auto.Pos[7].Pos := 270000;
   Auto.Pos[8].Pos := 315000;
   Auto.Pos[9..20].Pos := 0;
   Auto.Pos[1..8].Vel := 10000;
   Auto.Pos[9..20].Vel := 0;
   // Auto.Pos[1] : 1.取料位置
   // Auto.Pos[2] : 2.放料位置
   // Auto.Pos[3] : 3.
   // Auto.Pos[4] : 4.
   // Auto.Pos[5] : 5.
   // Auto.Pos[6] : 6.
   // Auto.Pos[7] : 7.
   // Auto.Pos[8] : 8.
   // Auto.Pos[9] : 9.
   PositionOk[1] := FALSE;   // [1]
   PositionOk[2] := FALSE;   // [2]
   PositionOk[3] := FALSE;   // [3]
   PositionOk[4] := FALSE;   // [4]
   PositionOk[5] := FALSE;   // [5]
   PositionOk[6] := FALSE;   // [6]
   PositionOk[7] := FALSE;   // [7]
   PositionOk[8] := FALSE;   // [8]
   PositionOk[9] := FALSE;   // [9]
   PositionOk[10..20] := FALSE;
END_DATA_BLOCK

DATA_BLOCK "ServoV90_A3"   // DB2503
{ S7_Optimized_Access := 'FALSE' }
// stored: AutoNumber false
   VAR
      In : Struct
         iInterlock : Bool := TRUE;   // interlock
         "iManJog+" : Bool := FALSE;   // positive motion/action/...manually
         "iManJog-" : Bool := FALSE;   // negtive motion/action/...manually
         iAutoStart : Bool := FALSE;   // negtive motion/action/...automaticly
         iHome : Bool := FALSE;   // Homing
         iCancelTask : Bool := FALSE;   // Cancel task
         iPauseTask : Bool := FALSE;   // Pause task
         iManStart : Bool := FALSE;   // positive motion/action/...automaticly
         iManListStart : Bool := FALSE;
         iLimitSwitchActive : Bool := TRUE;
         iLimitSoftActive : Bool := TRUE;
         iRunningTimeout : Time := T#0MS;
         iHomingTimeout : Time := T#0MS;
         iAutoPosition : DInt := 0;
         iAutoVelocity : Int := 0;
         iManListPosition : DInt := 0;
         iManListVelocity : Int := 0;
         iManListNumber : Int := 0;   // position list number
         iManPosition : DInt := 0;
         iManVelocity : Int := 0;
         iMode : Int := 0;   // 1-相对;2-绝对
      END_STRUCT;
      Out : Struct
         oReady : Bool := FALSE;
         oWarning : Bool := FALSE;   // warning
         oError : Bool := TRUE;   // error
         oInterlock : Bool := TRUE;
         oServoEnable : Bool := FALSE;
         oRunning : Bool := FALSE;
         oHoming : Bool := FALSE;
         oHomeRef : Bool := TRUE;
         oServoPosOK : Bool := FALSE;
         oErrorCode : Int := -244;
         oStatus : Int := 0;
         oActPosition : DInt := -3;
         oManualListPos : DInt := 0;
      END_STRUCT;
      IO : Struct
         ioManEnale : Bool := FALSE;
         ioAutoEnale : Bool := FALSE;
         ioAutoHome : Bool;
      END_STRUCT;
      Spare : Struct
         S : Array[0..100] of Byte;
      END_STRUCT;
      Manual : Struct
         Index : Int := 1;
         Pos : Array[1..20] of Struct
            Pos : DInt;
            Vel : Int;
         END_STRUCT;
      END_STRUCT;
      Auto : Struct
         Index : Int := 1;
         Pos : Array[1..20] of Struct
            Pos : DInt;
            Vel : Int;
         END_STRUCT;
      END_STRUCT;
      Interlock : Struct
         Active : Bool := FALSE;
         Case1 : Bool := TRUE;
         Case2 : Bool := TRUE;
         Case3 : Bool := FALSE;
         Case4 : Bool := FALSE;
         Case5 : Bool := FALSE;
         Case6 : Bool := FALSE;
         Case7 : Bool := FALSE;
         Case8 : Bool := FALSE;
         Case9 : Bool := FALSE;
         Case10 : Bool := FALSE;
      END_STRUCT;
      PositionOk : Array[1..20] of Bool;
      Home_Pos : Struct
         "Home Pos Pls" : Bool := FALSE;
         "Arrow indication" : Int := 0;
         "Process prompt" : Int := 0;
         "Button prompt" : Int := 0;
      END_STRUCT;
   END_VAR
BEGIN
   Spare.S[0..100] := 16#00;
   Manual.Pos[1].Pos := 0;
   Manual.Pos[2..6].Pos := 680000;
   Manual.Pos[7].Pos := 90000;
   Manual.Pos[8].Pos := 180000;
   Manual.Pos[9].Pos := 270000;
   Manual.Pos[10..20].Pos := 0;
   Manual.Pos[1].Vel := 20000;
   Manual.Pos[2..9].Vel := 10000;
   Manual.Pos[10..20].Vel := 0;
   Auto.Pos[1].Pos := 0;
   Auto.Pos[2..6].Pos := 680000;
   Auto.Pos[7].Pos := 90000;
   Auto.Pos[8].Pos := 180000;
   Auto.Pos[9].Pos := 270000;
   Auto.Pos[10..20].Pos := 0;
   Auto.Pos[1].Vel := 20000;
   Auto.Pos[2..9].Vel := 10000;
   Auto.Pos[10..20].Vel := 0;
   // Auto.Pos[1] : 1.取料位置
   // Auto.Pos[2] : 2.放料位置
   // Auto.Pos[3] : 3.
   // Auto.Pos[4] : 4.
   // Auto.Pos[5] : 5.
   // Auto.Pos[6] : 6.
   // Auto.Pos[7] : 7.
   // Auto.Pos[8] : 8.
   // Auto.Pos[9] : 9.
   PositionOk[1] := FALSE;   // [1]
   PositionOk[2] := FALSE;   // [2]
   PositionOk[3] := FALSE;   // [3]
   PositionOk[4] := FALSE;   // [4]
   PositionOk[5] := FALSE;   // [5]
   PositionOk[6] := FALSE;   // [6]
   PositionOk[7] := FALSE;   // [7]
   PositionOk[8] := FALSE;   // [8]
   PositionOk[9] := FALSE;   // [9]
   PositionOk[10..20] := FALSE;
END_DATA_BLOCK

DATA_BLOCK "ServoV90_A4"   // DB2504
{ S7_Optimized_Access := 'FALSE' }
// stored: AutoNumber false
   VAR
      In : Struct
         iInterlock : Bool := TRUE;   // interlock
         "iManJog+" : Bool := FALSE;   // positive motion/action/...manually
         "iManJog-" : Bool := FALSE;   // negtive motion/action/...manually
         iAutoStart : Bool := FALSE;   // negtive motion/action/...automaticly
         iHome : Bool := FALSE;   // Homing
         iCancelTask : Bool := FALSE;   // Cancel task
         iPauseTask : Bool := FALSE;   // Pause task
         iManStart : Bool := FALSE;   // positive motion/action/...automaticly
         iManListStart : Bool := FALSE;
         iLimitSwitchActive : Bool := TRUE;
         iLimitSoftActive : Bool := TRUE;
         iRunningTimeout : Time := T#0MS;
         iHomingTimeout : Time := T#0MS;
         iAutoPosition : DInt := 0;
         iAutoVelocity : Int := 0;
         iManListPosition : DInt := 0;
         iManListVelocity : Int := 0;
         iManListNumber : Int := 0;   // position list number
         iManPosition : DInt := 0;
         iManVelocity : Int := 0;
         iMode : Int := 0;   // 1-相对;2-绝对
      END_STRUCT;
      Out : Struct
         oReady : Bool := FALSE;
         oWarning : Bool := FALSE;   // warning
         oError : Bool := TRUE;   // error
         oInterlock : Bool := TRUE;
         oServoEnable : Bool := FALSE;
         oRunning : Bool := FALSE;
         oHoming : Bool := FALSE;
         oHomeRef : Bool := TRUE;
         oServoPosOK : Bool := FALSE;
         oErrorCode : Int := -244;
         oStatus : Int := 0;
         oActPosition : DInt := 260748;
         oManualListPos : DInt := 3585;
      END_STRUCT;
      IO : Struct
         ioManEnale : Bool := FALSE;
         ioAutoEnale : Bool := FALSE;
      END_STRUCT;
      Spare : Struct
         S : Array[0..100] of Byte;
      END_STRUCT;
      Manual : Struct
         Index : Int := 1;
         Pos : Array[1..20] of Struct
            Pos : DInt;
            Vel : Int;
         END_STRUCT;
      END_STRUCT;
      Auto : Struct
         Index : Int := 7;
         Pos : Array[1..20] of Struct
            Pos : DInt;
            Vel : Int;
         END_STRUCT;
      END_STRUCT;
      Interlock : Struct
         Active : Bool := FALSE;
         Case1 : Bool := TRUE;
         Case2 : Bool := TRUE;
         Case3 : Bool := FALSE;
         Case4 : Bool := FALSE;
         Case5 : Bool := FALSE;
         Case6 : Bool := FALSE;
         Case7 : Bool := FALSE;
         Case8 : Bool := FALSE;
         Case9 : Bool := FALSE;
         Case10 : Bool := FALSE;
      END_STRUCT;
      PositionOk : Array[1..20] of Bool;
      Home_Pos : Struct
         "Home Pos Pls" : Bool := FALSE;
         "Arrow indication" : Int := 0;
         "Process prompt" : Int := 0;
         "Button prompt" : Int := 0;
      END_STRUCT;
   END_VAR
BEGIN
   Spare.S[0..100] := 16#00;
   Manual.Pos[1].Pos := 3585;
   Manual.Pos[2].Pos := 48610;
   Manual.Pos[3].Pos := 93637;
   Manual.Pos[4].Pos := 138606;
   Manual.Pos[5].Pos := 183388;
   Manual.Pos[6].Pos := 228458;
   Manual.Pos[7].Pos := 273513;
   Manual.Pos[8].Pos := 318501;
   Manual.Pos[9..20].Pos := 0;
   Manual.Pos[1..8].Vel := 10000;
   Manual.Pos[9..20].Vel := 0;
   Auto.Pos[1].Pos := 3585;
   Auto.Pos[2].Pos := 48610;
   Auto.Pos[3].Pos := 93637;
   Auto.Pos[4].Pos := 138606;
   Auto.Pos[5].Pos := 183388;
   Auto.Pos[6].Pos := 228458;
   Auto.Pos[7].Pos := 273513;
   Auto.Pos[8].Pos := 318501;
   Auto.Pos[9..20].Pos := 0;
   Auto.Pos[1..8].Vel := 10000;
   Auto.Pos[9..20].Vel := 0;
   // Auto.Pos[1] : 1.取料位置
   // Auto.Pos[2] : 2.放料位置
   // Auto.Pos[3] : 3.
   // Auto.Pos[4] : 4.
   // Auto.Pos[5] : 5.
   // Auto.Pos[6] : 6.
   // Auto.Pos[7] : 7.
   // Auto.Pos[8] : 8.
   // Auto.Pos[9] : 9.
   PositionOk[1] := FALSE;   // [1]
   PositionOk[2] := FALSE;   // [2]
   PositionOk[3] := FALSE;   // [3]
   PositionOk[4] := FALSE;   // [4]
   PositionOk[5] := FALSE;   // [5]
   PositionOk[6] := FALSE;   // [6]
   PositionOk[7] := FALSE;   // [7]
   PositionOk[8] := FALSE;   // [8]
   PositionOk[9] := FALSE;   // [9]
   PositionOk[10..20] := FALSE;
END_DATA_BLOCK

DATA_BLOCK "ServoV90_DeviceCtl"   // DB4073
{ S7_Optimized_Access := 'FALSE' }
// stored: AutoNumber false
   VAR RETAIN
      V90Servo : Array[1..4] of Struct
         i : Int;
         nError : Int;
         nWarning : Int;
         nPositionListNo : Int;
         Pos : "PosList";
         Point : Array[0..39] of Struct
            Start : Bool;
            Achieve : Bool;
         END_STRUCT;
      END_STRUCT;
   END_VAR
BEGIN
   V90Servo[1..4].nPositionListNo := 1;
   // V90Servo[1].Pos.List[1] : 待机位
   // V90Servo[1].Pos.List[2] : 排钉位
   // V90Servo[1].Pos.List[3] : 第一个颗螺钉位置
   // V90Servo[1].Pos.List[4] : 第二个颗螺钉位置
   // V90Servo[2].Pos.List[1] : 待机位
   // V90Servo[2].Pos.List[2] : 排钉位
   // V90Servo[2].Pos.List[3] : 第一个颗螺钉位置
   // V90Servo[2].Pos.List[4] : 第二个颗螺钉位置
   V90Servo[1].Pos.List[4..19].Pos := 0;
   V90Servo[1].Pos.List[3..19].Vel := 0;
   // V90Servo[1].Point[1] : 初始位 / 上料位1
   // V90Servo[1].Point[2] : 抓料位 / 上料位2
   // V90Servo[1].Point[3] : 上料拍照位 / 上料位3
   // V90Servo[1].Point[4] : 下料位1 / 上料位4
   // V90Servo[1].Point[5] : 下料位2 / 上料位5
   // V90Servo[1].Point[6] : 下料位3 / 上料位6
   // V90Servo[1].Point[7] : 下料位4 / 上料位7
   // V90Servo[1].Point[8] : 下料位5 / 上料位8
   // V90Servo[1].Point[9] : NG下料位
   // V90Servo[2].Point[1] : 初始位
   // V90Servo[2].Point[2] : 取料位1 / 扫码位置2
   // V90Servo[2].Point[3] : 取料位2 / 扫码位置3
   // V90Servo[2].Point[4] : 取料位3 / 扫码位置4
   // V90Servo[2].Point[5] : 取料位4 / 扫码位置5
   // V90Servo[2].Point[6] : 取料位5 / 扫码位置6
   // V90Servo[2].Point[7] : 清洁位 / 扫码位置7
   // V90Servo[2].Point[8] : NG位 / 扫码位置8
   // V90Servo[2].Point[9] : 快速装配位
   // V90Servo[2].Point[10] : 慢速装配位
END_DATA_BLOCK

DATA_BLOCK "ST10_DBInterface_Stopper"   // DB2602
{ S7_Optimized_Access := 'FALSE' }
// stored: AutoNumber false
   VAR
      Stopper { S7_SetPoint := 'True'} : Array[1..50] of "UDT_StopperInterface";
   END_VAR
BEGIN
END_DATA_BLOCK

